PID_Status();
R_TRIG_0(CLK := PID.MODE.eMode=ePID_Modes.Auto); // R_trig
IF R_TRIG_0.Q THEN _w1 := PID.HMI_Target; END_IF
PID.PLC_Target := _w1;
_w2 := SEL(PID.MODE.eMode=ePID_Modes.Auto, PId.HMI_Target, PID.PLC_Target);
PID.Live_Target := _w2;
_w3 := _w2 * PID.FF;
PID.CV_FF := _w3;
_w4 := SEL(Reverse, _w2 - PID.Actual, PID.Actual - _w2);
PID.Err := _w4;
_w5 := SEL(PID.MODE.eMode=ePID_Modes.Auto, PID.MODE.eMode=ePID_Modes.FORCED_ON, PID.PLC_Enable AND (Not(PID.Inhibit))) AND True AND CV_OK AND PV_OK;
Loop_Enable := _w5;
FT_PIDW_0(
    IN := _w4,
    KP := PID.KP,
    TN := PID.TN,
    TV := PID.TV,
    LIM_L := PID.CV_Min-PID.CV_FF,
    LIM_H := PID.CV_Max-PID.CV_FF,
    RST := R_Trig_1.Q OR NOT _w5); // BURKERT_OSCAT_BASIC.FT_PIDW
_w6 := SEL(Loop_Enable, PID.CV_Min, _w3 + FT_PIDW_0.Y);
CV := _w6;
PID.CV := _w6;
PID.CV_P := PID.Err * PID.KP;
PID.CV_I := FT_PIDW_0.YI;
PID.CV_D := FT_PIDW_0.diff.out;
PID.Ready := (PID.MODE.eMode=ePID_Modes.Auto) AND CV_OK AND PV_OK;
R_TRIG_1(CLK := (PID.CV_P>0) AND (PID.CV_I<0) AND (FT_PIDW_0.Y<0.5) AND _w5); // R_Trig
IF NOT (PID.MODE.eMode=ePID_Modes.FORCED_ON) THEN _w7 := PID.PLC_Target; END_IF
PID.HMI_Target := _w7;

END_FUNCTION_BLOCK

// 20 Program Organization Units/Level_2_Controls/Quick_Mix_UDFB
FUNCTION_BLOCK Quick_Mix_UDFB
VAR_INPUT
	Destination_OK:BOOL;
END_VAR
VAR_OUTPUT
	//Active:BOOL;
	OK:BOOL;
END_VAR
VAR
	Current_Mode:eQuick_Mix_modes;
	Current_Status:eQuick_Mix_Status;
	SFCReset:BOOL;
	SFCInit:BOOL;
	PLC_Active:BOOL;
	Temp_PID:BURKERT_OSCAT_BASIC.FT_PIDW;
	Flow_PID:BURKERT_OSCAT_BASIC.FT_PIDW;
	Ramp:Burkert_OSCAT_BASIC.SRAMP;
	tRamp:Burkert_OSCAT_BASIC.SRAMP;
	Ramp_Time:TIME;
	Pause_Active:BOOL;
	Pause_Ton:Ton;
	//Temp_Control:Burkert_OSCAT_BASIC.SCALE_R;
	//Flow_Control:Burkert_OSCAT_BASIC.SCALE_R;
	tHW:REAL;
END_VAR
VAR_IN_OUT
	HW:cACV;
	CW:cACV;
	FIT:cFIT;
	TT:cAIT;
	Loop:Quick_Mix_Dut;
END_VAR

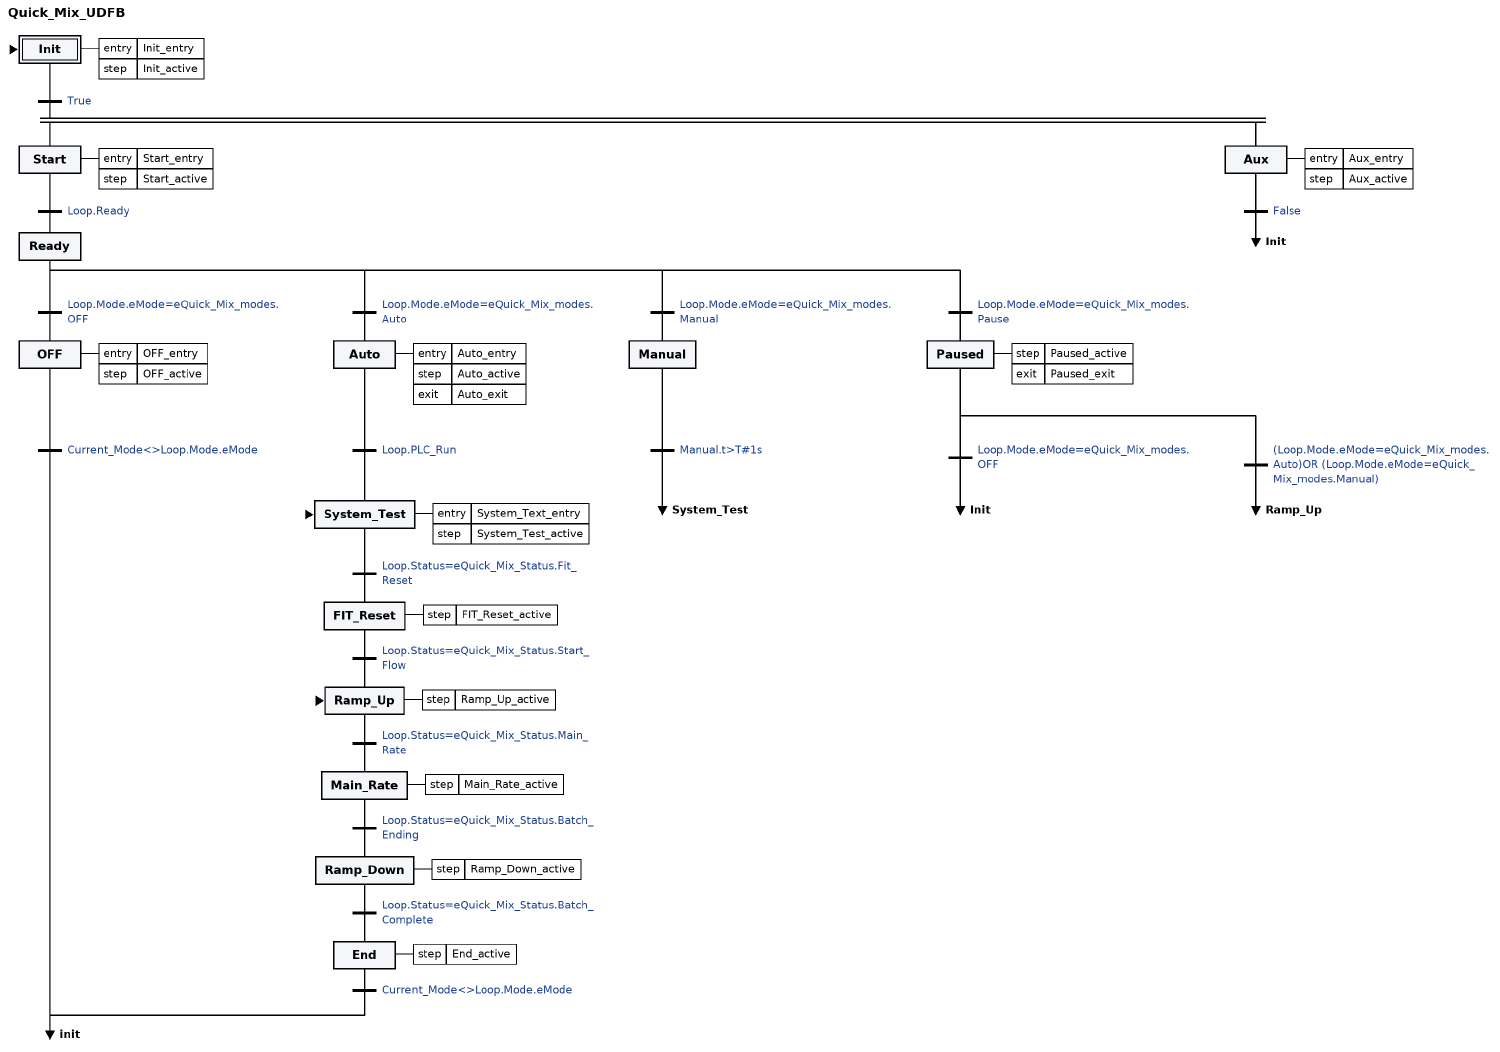
INITIAL_STEP Init:
    Init_entry(P1);  // entry action
    Init_active(N);  // step action
END_STEP
TRANSITION FROM Init TO (Start, Aux)
    := True;
END_TRANSITION
STEP Start:
    Start_entry(P1);  // entry action
    Start_active(N);  // step action
END_STEP
TRANSITION FROM Start TO Ready
    := Loop.Ready;
END_TRANSITION
STEP Ready:
END_STEP
STEP Aux:
    Aux_entry(P1);  // entry action
    Aux_active(N);  // step action
END_STEP
TRANSITION FROM Aux TO Init
    := False;
END_TRANSITION
TRANSITION FROM Ready TO OFF
    := Loop.Mode.eMode=eQuick_Mix_modes.OFF;
END_TRANSITION
STEP OFF:
    OFF_entry(P1);  // entry action
    OFF_active(N);  // step action
END_STEP
TRANSITION FROM OFF TO init
    := Current_Mode<>Loop.Mode.eMode;
END_TRANSITION
TRANSITION FROM Ready TO Auto
    := Loop.Mode.eMode=eQuick_Mix_modes.Auto;
END_TRANSITION
STEP Auto:
    Auto_entry(P1);  // entry action
    Auto_active(N);  // step action
    Auto_exit(P0);  // exit action
END_STEP
TRANSITION FROM Auto TO System_Test
    := Loop.PLC_Run;
END_TRANSITION
STEP System_Test:
    System_Text_entry(P1);  // entry action
    System_Test_active(N);  // step action
END_STEP
TRANSITION FROM System_Test TO FIT_Reset
    := Loop.Status=eQuick_Mix_Status.Fit_Reset;
END_TRANSITION
STEP FIT_Reset:
    FIT_Reset_active(N);  // step action
END_STEP
TRANSITION FROM FIT_Reset TO Ramp_Up
    := Loop.Status=eQuick_Mix_Status.Start_Flow;
END_TRANSITION
STEP Ramp_Up:
    Ramp_Up_active(N);  // step action
END_STEP
TRANSITION FROM Ramp_Up TO Main_Rate
    := Loop.Status=eQuick_Mix_Status.Main_Rate;
END_TRANSITION
STEP Main_Rate:
    Main_Rate_active(N);  // step action
END_STEP
TRANSITION FROM Main_Rate TO Ramp_Down
    := Loop.Status=eQuick_Mix_Status.Batch_Ending;
END_TRANSITION
STEP Ramp_Down:
    Ramp_Down_active(N);  // step action
END_STEP
TRANSITION FROM Ramp_Down TO End
    := Loop.Status=eQuick_Mix_Status.Batch_Complete;
END_TRANSITION
STEP End:
    End_active(N);  // step action
END_STEP
TRANSITION FROM End TO init
    := Current_Mode<>Loop.Mode.eMode;
END_TRANSITION
TRANSITION FROM Ready TO Manual
    := Loop.Mode.eMode=eQuick_Mix_modes.Manual;
END_TRANSITION
STEP Manual:
END_STEP
TRANSITION FROM Manual TO System_Test
    := Manual.t>T#1s;
END_TRANSITION
TRANSITION FROM Ready TO Paused
    := Loop.Mode.eMode=eQuick_Mix_modes.Pause;
END_TRANSITION
STEP Paused:
    Paused_active(N);  // step action
    Paused_exit(P0);  // exit action
END_STEP
TRANSITION FROM Paused TO Init
    := Loop.Mode.eMode=eQuick_Mix_modes.OFF;
END_TRANSITION
TRANSITION FROM Paused TO Ramp_Up
    := (Loop.Mode.eMode=eQuick_Mix_modes.Auto)OR (Loop.Mode.eMode=eQuick_Mix_modes.Manual);
END_TRANSITION

END_FUNCTION_BLOCK

// 20 Program Organization Units/Level_2_Controls/Rate_Batch
FUNCTION_BLOCK Rate_Batch
VAR_INPUT
	Config: REFERENCE TO cBatch;
	Rate_PID:	REFERENCE TO PID_Control;
	Volume_PID:	REFERENCE TO PID_Control;
	FIT:	REFERENCE TO cFIT;
	
	CV_OK:BOOL;
END_VAR
VAR_OUTPUT
	CV:REAL;
END_VAR
VAR
	Local_Mode:eHOA_Modes;
	Local_Task:eBatch_Task;
	Local_Status:eBatch_Status;
	
	Start_Rate:REAL;
	Main_Rate:REAL;
	End_Rate:REAL;
	
	
	Batch_Duration_S:UINT;
	clk_250:Burkert_OSCAT_BASIC.CLK_PRG;
	Batch_Clock_S:REAL;
	
END_VAR

CASE Config.Mode.eMode OF
	eHOA_Modes.Off:		Mode_OFF();
	eHOA_Modes.Manual:	Mode_Manual();
	eHOA_Modes.Auto:	Mode_Auto();	
END_CASE


CASE Config.Task OF
	eBatch_task.OFF	: 	Task_OFf();
	eBatch_task.Pause :	Task_Pause();
	eBatch_Task.Resume: Task_Resume();
	eBatch_task.Run:	Task_Run();
END_CASE

END_FUNCTION_BLOCK

// 20 Program Organization Units/Level_2_Controls/SSR_Heater
FUNCTION_BLOCK SSR_Heater
VAR_INPUT
	Heater: REFERENCE TO cSSR_heater;
	CV:REAL;
END_VAR
VAR_OUTPUT
	
END_VAR
VAR
	//Output_CV:UINT;
	CV_Error:REAL;
	//Output_Base:UINT;
	//Output_Map:WORD;
	
	SRR_1_U_CTRL:OSCAT_BUILDING.ACTUATOR_PUMP;
	SRR_1_V_CTRL:OSCAT_BUILDING.ACTUATOR_PUMP;
	SRR_1_W_CTRL:OSCAT_BUILDING.ACTUATOR_PUMP;
	
	SRR_2_U_CTRL:OSCAT_BUILDING.ACTUATOR_PUMP;
	SRR_2_V_CTRL:OSCAT_BUILDING.ACTUATOR_PUMP;
	SRR_2_W_CTRL:OSCAT_BUILDING.ACTUATOR_PUMP;
	
	SRR_3_U_CTRL:OSCAT_BUILDING.ACTUATOR_PUMP;
	SRR_3_V_CTRL:OSCAT_BUILDING.ACTUATOR_PUMP;
	SRR_3_W_CTRL:OSCAT_BUILDING.ACTUATOR_PUMP;
	
	Main_Contactor: RS;
	Force_Group_Sort:Bool;
	Group_Sorted:BOOL;
	Group_Sort_Array:ARRAY[0..2] OF REAL;
	Group_Sort_Index:ARRAY[0..2] OF INT;
	

	Pulse_30Min:Burkert_OSCAT_BASIC.CLK_PRG;
	CV_Index:INT:=0;
	Ramp:util.RAMP_REAL;
END_VAR

(*

0%			ALL OFF
11%			Single Pair
22%			2 Single Pair 
33%			Double Pair Full SSR
44%			Double Pair plus Single
55%			Double Pair Plus 2 Single Pairs
66%			2 Double Pair Full SSR
77%			Double Pair Full SSR + Single Pair
88%			
99%			All SSR's
*)



Select_CV();
Pulse_30Min(PT:=T#30M);
IF Pulse_30Min.Q OR Force_Group_Sort THEN
	Sort_Groups();
END_IF;

Set_Ouputs();

//Outputs();

SSR_Control();

RAMP( 
	ASCEND:= 10, 
	DESCEND:= 10, 
	TIMEBASE:= T#10S, 
	RESET:= , 
	OUT=>Heater.Effective_Output );

END_FUNCTION_BLOCK

// 20 Program Organization Units/Level_2_Controls/Stack_Lights_4Way
FUNCTION_BLOCK Stack_Lights_4Way
VAR_INPUT
END_VAR
VAR_OUTPUT
	Red:BOOL;
	Yellow:BOOL;
	Green:BOOL;
	Horn:BOOL;
	
END_VAR
VAR
	
	GEN_PULSE_RED: Burkert_OSCAT_BASIC.GEN_PULSE;
	GEN_PULSE_Yellow: Burkert_OSCAT_BASIC.GEN_PULSE;
	GEN_PULSE_Green: Burkert_OSCAT_BASIC.GEN_PULSE;
	GEN_PULSE_Horn: Burkert_OSCAT_BASIC.GEN_PULSE;
END_VAR

VAR_IN_out
	Device:c4Way_Stack_Light;
END_VAR
VAR // added by the converter: edge detectors and wires of the graphical bodies
    _w1, _w2, _w3, _w4 : ANY;
END_VAR

GEN_PULSE_Yellow(
    ENQ := Device.Yellow.Flash_Rate_ms>500 AND Device.Yellow.ON,
    PTH := To_Time(Device.Yellow.Flash_Rate_ms),
    PTL := To_Time(Device.Yellow.Flash_Rate_ms)); // Burkert_OSCAT_BASIC.GEN_PULSE
GEN_PULSE_Green(
    ENQ := Device.Green.Flash_Rate_ms>500 AND Device.Green.ON,
    PTH := To_Time(Device.Green .Flash_Rate_ms),
    PTL := To_Time(Device.Green .Flash_Rate_ms)); // Burkert_OSCAT_BASIC.GEN_PULSE
GEN_PULSE_Horn(
    ENQ := Device.Horn.Flash_Rate_ms>500 AND Device.Horn.ON,
    PTH := To_Time(Device.Horn .Flash_Rate_ms),
    PTL := To_Time(Device.Horn .Flash_Rate_ms)); // Burkert_OSCAT_BASIC.GEN_PULSE
_w1 := Device.Horn.ON AND NOT GEN_PULSE_Horn.Q;
Horn := _w1;
_w2 := Device.Yellow.ON AND NOT GEN_PULSE_Yellow.Q;
Device.Yellow.Q := _w2;
Yellow := _w2;
_w3 := Device.Green.ON AND NOT GEN_PULSE_Green.Q;
Device.Green.Q := _w3;
Green := _w3;
GEN_PULSE_RED(
    ENQ := Device.RED.Flash_Rate_ms>500 AND Device.RED.ON,
    PTH := To_Time(Device.RED.Flash_Rate_ms),
    PTL := To_Time(Device.RED.Flash_Rate_ms)); // Burkert_OSCAT_BASIC.GEN_PULSE
_w4 := Device.RED.ON AND NOT GEN_PULSE_RED.Q;
Device.RED.Q := _w4;
Red := _w4;
Device.Horn.Q := _w1;

END_FUNCTION_BLOCK

// 20 Program Organization Units/Level_2_Controls/SW_CTRL
FUNCTION_BLOCK SW_CTRL 
VAR_INPUT
	SW: REFERENCE TO cBatch_Transfer;
	FIT:REFERENCE TO cFIT;
	BCV:REFERENCE TO cBCV;
	Pump_Ready:BOOL;
	Interlock:BOOL;
END_VAR
VAR
	PID: BURKERT_OSCAT_BASIC.FT_PIDW;
END_VAR

IF (
		((SW.Auto_Batch = FALSE AND SW.Mode.eMode=eBatch_Transfer_Mode.Auto) OR
		(SW.Mode.eMode=eBatch_Transfer_Mode.Disabled)) AND SW.Status<> Transfer_Status.IDLE
	) THEN
	SW.Status:=Transfer_Status.IDLE;
END_IF;

IF (FIT.Rate.EU>1 AND NOT(BCV.Status.eStatus=eBCV_Status.A_Open) AND NOT(Interlock)) THEN
	SW.Status:=Transfer_Status.Flow_Meter_Active;
	SW.Ready:=FALSE;
	SW.Active:=FALSE;
END_IF;

IF NOT(Pump_Ready) THEN
	SW.Status:=Transfer_Status.Pump_Not_Ready;
	SW.Ready:=FALSE;
	SW.Active:=FALSE;
END_IF


IF NOT(BCV.Ready) THEN
	SW.Status:=Transfer_Status.BCV_Not_Ready;
	SW.Ready:=FALSE;
	SW.Active:=FALSE;
END_IF;

IF (BCV.Status.eStatus=eBCV_Status.Interlocked OR BCV.Status.eStatus=eBCV_Status.LOCKED_OUT ) THEN
	SW.Status:=Transfer_Status.LOCKED_OUT;
	SW.Ready:=FALSE;
	SW.Active:=FALSE;
END_IF;


IF Sw.Status=Transfer_Status.IDLE AND Interlock THEN
	SW.Status:=Transfer_Status.LOCKED_OUT;
END_IF

CASE SW.Status OF
	
	Transfer_Status.IDLE:
		SW.Ready:=TRUE;
		SW.BCV:=FALSE;
		
		SW.Remaining_Time_S:=0;
		SW.Current_Rate:=0;
		SW.Current_Volume:=0;
		SW.Remaining_Volume:=0;
		SW.Active:=FALSE;
		
		IF (
			(SW.Auto_Batch AND SW.Mode.eMode=eBatch_Transfer_Mode.Auto) OR
			( SW.Mode.eMode=eBatch_Transfer_Mode.Batch)
			)THEN
			SW.Status:=Transfer_Status.FIT_Reset;
		END_IF;
		
		
	Transfer_Status.FIT_Reset:
		SW.Active:=TRUE;
		SW.BCV:=FALSE;
		SW.Remaining_Time_S:=0;
		FIT.PLC_Reset:=(FIT.Total>1);
		IF FIT.Total<1 THEN
			SW.Status:=Transfer_Status.Open_Valve;
		END_IF;
		
	Transfer_Status.Open_Valve:
	SW.BCV:=TRUE;
	IF SW.BCV AND BCV.Status.eStatus=eBCV_Status.A_Open THEN
			SW.Status:=Transfer_Status.Flow_Active;	
		END_IF;
		
	
		
	Transfer_Status.Flow_Active:
		SW.BCV:=TRUE;
		SW.Remaining_Time_S:=TO_UDINT(SW.Remaining_Volume/(FIT.Rate.EU/60));
		SW.Current_Rate:=FIT.Rate.EU;
		SW.Current_Volume:=FIT.Total;
		SW.Remaining_Volume:=(SW.Volume-FIT.Total);
		
		
		IF (
			(FIT.Rate.EU > (SW.Rate*0.25)) OR
			(FIT.Total> (SW.Volume*0.80))
		) THEN
			SW.Status:=Transfer_Status.Running;
		END_IF;
	Transfer_Status.Running:	
			SW.BCV:=TRUE;
			SW.Remaining_Time_S:=TO_UDINT(SW.Remaining_Volume/(FIT.Rate.EU/60));
			SW.Current_Rate:=FIT.Rate.EU;
			SW.Current_Volume:=FIT.Total;	
			SW.Remaining_Volume:=(SW.Volume-FIT.Total);
			IF (FIT.Total> SW.Volume)
			THEN
				SW.Status:=Transfer_Status.Complete;
			END_IF;
	Transfer_Status.Complete:
		SW.BCV:=FALSE;
		SW.Remaining_Time_S:=0;
		SW.Current_Rate:=0;
		SW.Current_Volume:=0;
		SW.Remaining_Volume:=0;
		SW.Active:=FALSE;
		
	Transfer_Status.LOCKED_OUT:
		SW.Ready:=FALSE;
		SW.Active:=FALSE;
		SW.Remaining_Time_S:=0;
		SW.Current_Rate:=0;
		SW.Current_Volume:=0;
		SW.Remaining_Volume:=0;
		
		
	Transfer_Status.Destination_Not_Ready:
		SW.Active:=FALSE;
		IF SW.BCV AND BCV.Status.eStatus=eBCV_Status.A_Open THEN
			SW.Status:=Transfer_Status.Flow_Active;		
		END_IF;
		IF 	(
				NOT(SW.Mode.eMode=eBatch_Transfer_mode.Auto AND SW.Auto_Batch = TRUE) AND
				NOT(SW.Mode.eMode=eBatch_Transfer_mode.Batch) AND
				SW.BCV=TRUE
			)THEN
			SW.BCV:=FALSE;
		END_IF;
	Transfer_Status.Flow_Meter_Active:
		IF FIT.Rate.EU<0.5 THEN
			SW.Status:=Transfer_Status.IDLE;
		END_IF;
END_CASE;



PID(
	IN:= (SW.Rate-FIT.Rate.EU), 
	KP:= SW.Config.KP, 
	TN:= SW.Config.TN, 
	TV:= SW.Config.TV, 
	LIM_L:= 0, 
	LIM_H:= 100-(SW.Config.FF*SW.Rate), 
	RST:= NOT(SW.Active) OR NOT(BCV.Status.eStatus=eBCV_Status.A_Open) , 
	Y=> , 
	LIM=> );
	
IF NOT(SW.Active) THEN
	SW.ACV:=0;
	SW.BCV:=FALSE;
ELSE
	SW.ACV:=PID.Y+(SW.Config.FF*SW.Rate);

END_IF;

END_FUNCTION_BLOCK

// 20 Program Organization Units/Level_2_Controls/Tempered_Line_4_Valve
FUNCTION_BLOCK Tempered_Line_4_Valve
VAR_INPUT
	Config_DATA:REFERENCE TO cTempered_Line_Data;
	
	HW_Supply_TT:REFERENCE TO cSensor;
	CW_Supply_TT:REFERENCE TO cSensor;
	
	CW_Inlet_PT:REFERENCE TO cSensor;
	CW_Outlet_PT:REFERENCE TO cSensor;
	HW_Inlet_PT:REFERENCE TO cSensor;
	HW_Outlet_PT:REFERENCE TO cSensor;
	Combined_Temp:REFERENCE TO cSensor;
	
	HW_FIT:REFERENCE TO cFIT;
	CW_FIT:REFERENCE TO cFIT;

	HW_PID		:REFERENCE TO PID_DUT;
	CW_PID		:REFERENCE TO PID_DUT;
	Temperature_PID		:REFERENCE TO PID_DUT;
	
	CW1_ACV		:REFERENCE TO cACV;
	CW2_ACV		:REFERENCE TO cACV;
	HW1_ACV		:REFERENCE TO cACV;
	HW2_ACV		:REFERENCE TO cACV;
	
	KV_Curve	:REFERENCE TO ARRAY[0..100] OF REAL;
	CV_2_KV		:REFERENCE TO ARRAY[0..100] OF REAL;
	
	Temp_Flow_CV	:REFERENCE TO cTempered_C;
	
	Flow_Units:eUnits;
	Temperature_Units:eUnits;
	Run_mode:BYTE;
	
	
	HW_CV_Mode_3:INT;
	CW_CV_Mode_3:INT;
	
END_VAR
VAR_OUTPUT
END_VAR
VAR
	Local_Mode:eTempered_modes;
	Local_Task:eTempered_Task;
	Local_Status:eTempered_Status;
	On_Target:BOOL;
	Task_Ton:Ton;
	Prepare_TON:TON;
	
	
	Temp_Index:INT;
	Flow_Index:INT;
	
	CW_KV_Index:INT;
	HW_KV_Index:INT;
	
	CW_Target_KV_Index:INT;
	HW_Target_KV_Index:INT;
	
	Calibration_Temp:cAlarm_Window;
	
	
	KV_Index_Scalar:INT:=20;
	
	HW_CV_Ramp:RAMP_REAL;
	CW_CV_Ramp:RAMP_REAL;
	
	TOF_0: TOF;
END_VAR

AUX();
Alarms();
Math();
PID_CTRL();
ACV_CTRL();

Task_Ton();

END_FUNCTION_BLOCK

// 20 Program Organization Units/Level_2_Controls/Tempered_Mix_UDFB
FUNCTION_BLOCK Tempered_Mix_UDFB
VAR_INPUT
	//Loop_ID:INT;
END_VAR
VAR_IN_OUT
	HW_ACV:cACV;
	CW_ACV:cACV;
	Temperature:cAIT;
	FIT:cFIT;
	Control:Mix_DUT;
END_VAR
VAR_OUTPUT
END_VAR
VAR
	R_TRIG_0: R_Trig;
	RATE_PID: BURKERT_OSCAT_BASIC.CTRL_PID;
	
	Temp_PID: BURKERT_OSCAT_BASIC.CTRL_PID;
	TON_0: TON;
	Stage_Delay: TIME := T#2s;
	TON_1: TON;
	TON_2: TON;
	SRAMP_0: BURKERT_OSCAT_BASIC.SRAMP;
	TON_3: TON;
	TON_4: TON;
	Ramp_Active: BOOL;
	Ramp_Target: REAL;
	TON_5: TON;
	TON_6: TON;
	R_TRIG_1: R_trig;
	Ramp_Start_Volume: REAL;
	Ramp_Volume: REAL;
	R_TRIG_2: R_Trig;
	R_TRIG_3: R_Trig;
	PID_0: Util.PID;
	R_TRIG_4: R_Trig;
	R_TRIG_5:R_trig;
	
	Live_Rate: REAL;
END_VAR
VAR // added by the converter: edge detectors and wires of the graphical bodies
    _w1, _w2, _w3, _w4, _w5, _w6, _w10, _w12, _w13, _w14, _w15, _w16, _w18, _w19, _w21, _w23, _w25, _w30, _w32 : ANY;
    _w7, _w8, _w9, _w11, _w17, _w20, _w22, _w24, _w26, _w28, _w29, _w31, _w33 : BOOL;
    _w27 : REAL;
END_VAR

// note: 18 stored wires end on pins the file does not list and are not shown
IF NOT (HW_ACV.Mode.eMode=eACV_Modes.Auto) THEN _w1 := Mix_Status.HW_Valve_Not_Ready; END_IF
Control.Status := _w1;
IF NOT (CW_ACV.Mode.eMode=eACV_Modes.Auto) THEN _w2 := Mix_Status.CW_Valve_Not_Ready; END_IF
Control.Status := _w2;
Control.Actual_Rate_EU := FIT.Rate.EU;
_w3 := (Control.Mode=Mix_Modes.IDlE) OR (Control.STATUS>Mix_Status.Batch_Ending) OR (Control.Mode=Mix_Modes.Pause);
RATE_PID(
    ACT := FIT.Rate.EU,
    SET := Live_Rate,
    SUP := 0.1,
    OFS := 0.0,
    M_I := 0.0,
    MAN := _w3,
    RST := _w3,
    KP := Control.Config.Flow_KP,
    TN := Control.Config.Flow_TN,
    TV := Control.Config.Flow_TV,
    LL := 0,
    LH := 100.0); // BURKERT_OSCAT_BASIC.CTRL_PID
Control.Flow_CV := RATE_PID.Y;
R_TRIG_2(CLK := _w3 AND (Temperature.Mode.eMode<>AIT_Modes.Forced)); // R_Trig
IF R_TRIG_2.Q THEN _w4 := AIT_Modes.Alarms_Disabled; END_IF
Temperature.Mode.eMode := _w4;
Control.Actual_Temp_EU := Temperature.EU;
_w5 := (Control.Mode=Mix_Modes.IDlE) OR (Control.Mode=Mix_Modes.Rate_Only) OR (Control.STATUS>Mix_Status.Batch_Ending) OR (Control.STATUS=Mix_Status.Start_Flow) OR (Control.STATUS=Mix_Status.Fit_Reset) OR (Control.Mode=Mix_Modes.Pause);
PID_0(
    ACTUAL := Temperature.EU,
    SET_POINT := Control.Config.TARGET_C,
    KP := Control.Config.Temp_KP,
    TN := Control.Config.Temp_TN,
    TV := Control.Config.Temp_TV,
    Y_MANUAL := 0,
    Y_OFFSET := 0,
    Y_MIN := -100,
    Y_MAX := 100,
    MANUAL := _w5,
    RESET := _w5); // Util.PID
Control.Temp_CV := SEl(Control.Mode=Mix_Modes.Cold_Only, SEl(Control.Mode=Mix_Modes.Hot_Only, PID_0.Y, 100), -100);
SRAMP_0(
    X := Ramp_Target,
    A_UP := Control.Config.Ramp_Rate,
    A_DN := 0-Control.config.Ramp_Rate,
    VU_MAX := Control.config.Max_Flow,
    VD_MAX := 0-Control.config.Max_Flow,
    LIMIT_HIGH := Control.config.Max_Flow,
    LIMIT_LOW := Control.Config.Min_Flow,
    RST := Control.Mode=Mix_Modes.IDlE); // BURKERT_OSCAT_BASIC.SRAMP
Live_Rate := SRAMP_0.Y;
IF Control.Mode=Mix_Modes.IDlE THEN _w6 := Mix_Status.IDle; END_IF
Control.STATUS := _w6;
R_TRIG_0(CLK := (Control.Mode=Mix_Modes.Auto) OR (Control.Mode=Mix_Modes.Hot_Only) OR (Control.Mode=Mix_Modes.Cold_Only) OR (Control.Mode=Mix_Modes.Quick_Start)); // R_Trig
Control.STATUS := SEL(R_TRIG_0.Q, Control.STATUS, Mix_Status.Fit_Reset);
Control.Actual_Volume_EU := FIT.Total;
_w7 := Control.STATUS = Mix_Status.Fit_Reset;
_w8 := NOT (FIT.Total>0.1) AND _w7;
FIT.PLC_Reset := SEL(_w7 AND (FIT.Total>0.1), SEL(_w8, FIT.PLC_Reset, False), True);
_w9 := _w8;
IF _w9 THEN _w10 := Mix_Status.Start_Flow; END_IF
_w11 := _w9;
IF _w11 THEN _w12 := SEL(Control.Mode=Mix_Modes.Hot_Only, _w10, Mix_Status.Temperature_OK); END_IF
IF _w11 THEN _w13 := SEL(Control.Mode=Mix_Modes.Hot_Only, _w12, Mix_Status.Temperature_OK); END_IF
Control.STATUS := _w13;
_w14 := Control.Temp_CV / 100.0;
_w15 := LIMIT(0, Control.Flow_CV * (1.0 + _w14), 100);
Control.HW_CMD := _w15;
HW_ACV.PLC_CMD := _w15;
_w16 := LIMIT(0, Control.Flow_CV * (1.0 - _w14), 100);
Control.CW_CMD := _w16;
CW_ACV.PLC_CMD := _w16;
_w17 := Control.STATUS = Mix_Status.Start_Flow;
IF _w17 THEN _w18 := Control.Config.Min_Flow; END_IF
Ramp_Target := _w18;
TON_0(IN := _w17 AND (Control.Actual_Rate_EU > (Control.Config.Min_Flow*0.8) OR (Control.Mode=Mix_Modes.Quick_Start)), PT := Stage_Delay); // TON
Control.STATUS := SEL(TON_0.Q, Control.STATUS, Mix_Status.Flow_Detected);
TON_1(IN := Control.STATUS = Mix_Status.Flow_Detected, PT := Stage_Delay); // TON
R_TRIG_3(CLK := (Temperature.Mode.eMode<>AIT_Modes.Forced) AND TON_1.Q); // R_Trig
IF R_TRIG_3.Q THEN _w19 := TT_Modes.Active; END_IF
Temperature.Mode.iMode := _w19;
Control.STATUS := SEL(TON_1.Q, Control.STATUS, Mix_Status.Start_temperature);
Temperature.Alarm_Config.Setpoints.Hi_Hi_Alarm := Control.Config.TARGET_C+(Control.Config.TEMP_WINDOW*4);
Temperature.Alarm_Config.Setpoints.Hi_Warn := Control.Config.TARGET_C+(Control.Config.TEMP_WINDOW*2);
Temperature.Alarm_Config.Setpoints.Low_warn := Control.Config.TARGET_C-(Control.Config.TEMP_WINDOW*2);
Temperature.Alarm_Config.Setpoints.Low_Low_Alarm := Control.Config.TARGET_C-(Control.Config.TEMP_WINDOW*4);
TON_2(IN := Control.STATUS = Mix_Status.Start_temperature AND (Control.Actual_Temp_EU > (Control.Config.TARGET_C-Control.Config.TEMP_WINDOW) OR (Control.Mode=Mix_Modes.Quick_Start)), PT := Stage_Delay); // TON
Control.STATUS := SEL(TON_2.Q, Control.STATUS, Mix_Status.Temperature_OK);
TON_3(IN := Control.STATUS = Mix_Status.Temperature_OK, PT := Stage_Delay); // TON
Control.STATUS := SEL(TON_3.Q, Control.STATUS, Mix_Status.Foundation_Rate);
_w20 := Control.STATUS = Mix_Status.Foundation_Rate;
IF _w20 THEN _w21 := Control.Config.Foundation_Rate; END_IF
Ramp_Target := _w21;
Control.STATUS := SEL(_w20 AND (Control.Actual_Rate_EU >= (Control.Config.Foundation_Rate*0.9) OR (Control.Mode=Mix_Modes.Quick_Start)), Control.STATUS, Mix_Status.Foundation_Rate_OK);
TON_4(IN := Control.STATUS = Mix_Status.Foundation_Rate_OK AND (FIT.Total >= Control.Config.Foundation_Volume OR (Control.Mode=Mix_Modes.Quick_Start)), PT := Stage_Delay); // TON
Control.STATUS := SEL(TON_4.Q, Control.STATUS, Mix_Status.Foundation_Amount_Complete);
R_TRIG_5(CLK := Control.Mode=Mix_Modes.Resume); // R_trig
TON_5(IN := Control.STATUS = Mix_Status.Foundation_Amount_Complete, PT := Stage_Delay); // TON
Control.STATUS := SEL(R_TRIG_5.Q OR TON_5.Q, Control.STATUS, Mix_Status.Main_Rate);
_w22 := Control.STATUS = Mix_Status.Main_Rate;
R_TRIG_1(CLK := _w22); // R_trig
IF R_TRIG_1.Q THEN _w23 := Control.Actual_Volume_EU; END_IF
Ramp_Start_Volume := _w23;
_w24 := _w22;
IF _w24 THEN _w25 := Control.Config.TARGET_lpm; END_IF
Ramp_Target := _w25;
_w26 := _w24 AND Control.Actual_Rate_EU >= (Control.Config.TARGET_lpm*0.9);
Control.STATUS := SEL(_w26, Control.STATUS, Mix_Status.Main_Rate_OK);
IF _w26 THEN _w27 := Control.Actual_Volume_EU - Ramp_Start_Volume; END_IF
Ramp_Volume := _w27;
_w28 := Control.STATUS = Mix_Status.Main_Rate_OK;
TON_6(IN := _w28, PT := Stage_Delay); // TON
Control.STATUS := SEL(TON_6.Q, Control.STATUS, Mix_Status.Grain_Dispense);
_w29 := Control.STATUS = Mix_Status.Grain_Dispense;
IF _w29 THEN _w30 := Control.Config.TARGET_lpm; END_IF
Ramp_Target := _w30;
Control.STATUS := SEL(_w29 AND Control.Actual_Volume_EU >= (Control.Config.TARGET_L-Control.Config.Foundation_Volume), Control.STATUS, Mix_Status.Batch_Ending);
Control.Grain_ETA_S := REAL_TO_INT(((Control.Config.TARGET_L-Control.Config.Foundation_Volume) - Control.Actual_Volume_EU) / (Control.Actual_Rate_EU/60));
_w31 := Control.STATUS = Mix_Status.Batch_Ending;
IF _w31 THEN _w32 := Control.Config.Foundation_Rate; END_IF
Ramp_Target := _w32;
_w33 := (_w22 OR _w28 OR _w29 OR _w31) AND Control.Actual_Volume_EU >= Control.Config.TARGET_L;
Ramp_Active := SEl(_w33, Ramp_Active, FALSE);
Control.STATUS := SEL(_w33, Control.STATUS, Mix_Status.Batch_Complete);
// 0.1: input not connected

END_FUNCTION_BLOCK

// 20 Program Organization Units/Simulators/c8691_CanOpen_Sim
FUNCTION_BLOCK cDigital_BCV_CanOpen_Sim
VAR_INPUT
	BCV: REFERENCE TO cDigital_BCV;
END_VAR
VAR_OUTPUT
END_VAR
VAR
END_VAR

BCV.PDO.EndPositions.1:=BCV.PDO.Setpoint.0;
BCV.PDO.EndPositions.0:=NOT(BCV.PDO.Setpoint.0);
BCV.PDO.NamurStatus:=1;

END_FUNCTION_BLOCK

// 20 Program Organization Units/Simulators/c8694_CanOpen_Sim
FUNCTION cDigital_ACV_CanOpen_Sim
VAR_INPUT
END_VAR
VAR_OUTPUT
	//CanState:_3SCOS.DED.DEVICE_STATE;
END_VAR
VAR
	//Data:Bytes_Dword;
END_VAR
VAR_IN_OUT
	Device:cCanOpen_8694;
END_VAR


Device.PDO.NamurStatus:=1;

Device.PDO.CMD:=Device.PDO.CMDdigital;
Device.PDO.Pos:=Device.PDO.CMDdigital;

//CanState:=_3SCOS.DED.DEVICE_STATE.RUNNING;


Device.CanOpen.Device_State:=_3SCOS.DED.DEVICE_STATE.RUNNING;

END_FUNCTION

// 20 Program Organization Units/Simulators/CalculateMixedConductivity
FUNCTION CalculateMixedConductivity : Real
VAR_INPUT
    Stream_A_Rate        : REAL;  (* Flow rate of Stream A in liters per minute *)
    Stream_A_Conductivity: REAL;  (* Conductivity of Stream A in µS/cm *)
    Stream_B_Rate        : REAL;  (* Flow rate of Stream B in liters per minute *)
    Stream_B_Conductivity: REAL;  (* Conductivity of Stream B in µS/cm *)
END_VAR
VAR
    TotalFlowRate       : REAL;
    WeightedConductivity: REAL;
END_VAR

IF Stream_A_Rate>0.05 AND Stream_B_Rate>0.05 THEN
    TotalFlowRate := Stream_A_Rate + Stream_B_Rate;
    WeightedConductivity := ((Stream_A_Conductivity * Stream_A_Rate) + (Stream_B_Conductivity * Stream_B_Rate)) / TotalFlowRate;
    CalculateMixedConductivity := WeightedConductivity;
ELSE
	CalculateMixedConductivity :=MIN(Stream_A_Conductivity,Stream_B_Conductivity);
END_IF;

END_FUNCTION

// 20 Program Organization Units/Simulators/CanOpen_8694_Data_Sim
FUNCTION CanOpen_8694_Data_Sim
VAR_INPUT
END_VAR
VAR_OUTPUT
END_VAR
VAR
	//Data:Bytes_Dword;
END_VAR
VAR_IN_OUT
	Device:cCanOpen_8694;
END_VAR



Device.PDO.NamurStatus:=1;
Device.PDO.Pos:=Device.PDO.CMDdigital;
Device.CanOpen.Device_State:=_3SCOS.DED.DEVICE_STATE.DISABLED;

END_FUNCTION

// 20 Program Organization Units/Simulators/Contactor_Sim
FUNCTION_BLOCK Contactor_Sim
VAR_INPUT
	Device:Contactor_DUT;
END_VAR
VAR_OUTPUT
	FWD_Limit:BOOL;
	Rev_Limit:BOOL;
END_VAR
VAR
	tPos:INT;
	pulse: Burkert_OSCAT_BASIC.CLK_PRG;
END_VAR

Pulse(PT:=T#1S);

IF Pulse.Q THEN
	
	IF Device.Q2 AND tPos>0 THEN tPos:=tPos-1; END_IF;
	IF Device.Q1 AND tPos<100 THEN tPos:=tpos+1; END_IF;
END_IF;


FWD_Limit:=tPos<100;
Rev_Limit:=tPos>0;

END_FUNCTION_BLOCK

// 20 Program Organization Units/Simulators/Eaton_DM1_Sim
FUNCTION Eaton_DM1_Sim : ARRAY[0..10] OF WORD;
VAR_INPUT
	TX:ARRAY[0..10] OF WORD;
END_VAR
VAR
END_VAR

//Status_Word RX[0]
Eaton_DM1_Sim[0].0:=TRUE;	//VFD.Data.Drive_STATUS.Ready:=
Eaton_DM1_Sim[0].1:=TX[0].0;		//VFD.Data.Drive_STATUS.Run:=
Eaton_DM1_Sim[0].2:=TX[0].1;	//VFD.Data.Drive_STATUS.FWD:=



//General Status RX[1]

//Actual Speed RX[2]
IF TX[0].0 THEN
	Eaton_DM1_Sim[2]:=TX[2];	//VFD.Output_Pct:=
	Eaton_DM1_Sim[3]:=(TX[2]/6);		//vfd.Output_Hz:=TO_REAL(
ELSE
	Eaton_DM1_Sim[2]:=0;
	Eaton_DM1_Sim[3]:=0;
END_IF;

Eaton_DM1_Sim[9]:=6240;	//VFD.Data.DC_Link:=TO_REAL(

END_FUNCTION

// 20 Program Organization Units/Simulators/eDip_8412_Sim
FUNCTION eDip_8412_Sim : Bool
VAR_INPUT
	Current:REAL;
	Low_Limit:REAL;
	High_Limit:REAL;
	Rate_Up:REAL;
	Rate_Down:REAL;
END_VAR
VAR
	Data:Bytes_Dword;
END_VAR

VAR_OUTPUT
	RX_0:WORD;
	RX_1:WORD;
END_VAR

Data.tReal:=Current+(Rate_up-Rate_Down);
Data.tReal:=LIMIT(Low_limit,Data.tReal,High_Limit);

RX_0:=Data.tWord[1];
RX_1:=Data.tWord[0];

END_FUNCTION

// 20 Program Organization Units/Simulators/Edip_8691_Sim
FUNCTION Edip_8691_Sim
VAR_INPUT
	BCV: Reference to ceDip_8691;;
END_VAR
VAR_OUTPUT
END_VAR
VAR
END_VAR

//BCV.PDO.EndPositions.0:=BCV.PDO.Setpoint.0;
//BCV.PDO.EndPositions.1:=NOT(BCV.PDO.Setpoint.0);
//BCV.PDO.NamurStatus:=1;


(*
Join.tWord[0]:=BCV.RX[0];
BCV.PDO.EndPositions:=Join.tByte[1];

Join.tWord[0]:=BCV.RX[1];
BCV.PDO.NamurStatus:=Join.tByte[1];
Join.tWord[1]:=BCV.RX[2];
Join.tWord[0]:=BCV.RX[3];
BCV.PDO.Position:=Join.tReal;

Join.tByte[0]:=0;
Join.tByte[1]:=BCV.PDO.Setpoint;
BCV.TX:=Join.tWord[0];
*)

//BCV.RX[0].8:=BCV.TX.8;
//BCV.RX[0].9:=NOT(BCV.TX.8);
//BCV.RX[1]:=256;

END_FUNCTION

// 20 Program Organization Units/Simulators/Edip_8694_Data_Sim
FUNCTION Edip_8694_Data_Sim
VAR_INPUT
END_VAR
VAR_OUTPUT
END_VAR
VAR
	//Data:Bytes_Dword;
END_VAR
VAR_IN_OUT
	Device:ceDip_8694;
END_VAR


Device.RX.ActualPosition.tWord[0]:=Device.TX_CmdDigital.tWord[0];
Device.RX.ActualPosition.tWord[1]:=Device.TX_CmdDigital.tWord[1];

Device.RX.NamurStatus.tByte[1]:=1;

Device.RX.CurrentSetPoint.tWord[0]:=Device.TX_CmdDigital.tWord[0];
Device.RX.CurrentSetPoint.tWord[1]:=Device.TX_CmdDigital.tWord[1];


//Device.RX[5]:=0;

END_FUNCTION

// 20 Program Organization Units/Simulators/eDip_ME44_DI_Count_Sim
FUNCTION eDip_ME44_DI_Count_Sim : Bool
VAR_INPUT
	Pulse_250:BOOL;
	Rate_LPM:REAL;
	FIT:cFIT;
	//Current:REAL;
	
END_VAR
VAR
	//Data:Bytes_Dword;
END_VAR

VAR_OUTPUT
	Count:REAL;
END_VAR



IF NOT(FIT.PLC_Reset) AND NOT(FIT.HMI_Reset) THEN
	IF Pulse_250 THEN
		Count:=TO_REAL(FIT.Counts+(((Rate_LPM/60)/4)*FIT.K));
	ELSE
		Count:=TO_REAL(FIT.Counts);
	END_IF;
ELSE
	Count:=0;	
END_IF;

END_FUNCTION

// 20 Program Organization Units/Simulators/eDip_ME44_DI_Hz_Sim
FUNCTION eDip_ME44_DI_Hz_Sim : Bool
VAR_INPUT

	Rate_LPM:REAL;
	FIT:cFIT;
	
END_VAR
VAR
	//Data:Bytes_Dword;
	//Value:REAL;
END_VAR

VAR_OUTPUT
	Hz:Real;
END_VAR

IF NOT(FIT.PLC_Reset) AND NOT(FIT.HMI_Reset) THEN
	Hz:=(Rate_LPM/60)*FIT.K;
ELSE
	Hz:=0;	
END_IF;

END_FUNCTION

// 20 Program Organization Units/Simulators/FIT_Sim
FUNCTION FIT_Sim : UDINT
VAR_INPUT
	FIT: REFERENCE TO cFIT;
	Control:REAL;
	clk:Bool;
	
END_VAR
VAR_OUTPUT
	Hz:REAL;
END_VAR
VAR
	PLC_Time:UDINT;
END_VAR

IF FIT.HMI_Reset OR FIT.PLC_Reset THEN
	FIT.Counts:=0;
END_IF;

IF clk THEN	
	FIT.Counts:=(FIT.Counts + TO_UDINT(Control/4) );
	IF FIT.Counts=0 THEN FIT.Counts:=1; END_IF;
	
	
END_IF;
FIT_Sim:=FIT.Counts;
Hz:=(Control);

END_FUNCTION

// 20 Program Organization Units/Simulators/HTX_Sim
FUNCTION HTX_Sim : Bool
VAR_INPUT
    A_Rate      : REAL;  (* Mass flow rate of side A *)
    A_InletTemp : REAL;  (* Inlet temperature of side A *)
    B_Rate      : REAL;  (* Mass flow rate of side B *)
    B_InletTemp : REAL;  (* Inlet temperature of side B *)
END_VAR
VAR_OUTPUT
    A_OutletTemp : REAL; (* Outlet temperature of side A *)
    B_OutletTemp : REAL; (* Outlet temperature of side B *)
END_VAR
VAR
    Cp : REAL := 4.18;  (* Specific heat capacity (same for both sides) *)
END_VAR


   // A_OutletTemp := ((A_Rate * A_InletTemp) + (B_Rate * B_InletTemp)) / (A_Rate + B_Rate);
   /// B_OutletTemp := A_OutletTemp; 

    HTX_Sim := TRUE;
(*
IF A_Rate>0.1 THEN
		B_OutletTemp:=((A_Rate * A_InletTemp) + (B_Rate * B_InletTemp)) / (A_Rate + B_Rate);
ELSE	
		A_OutletTemp:= LIMIT(0,A_InletTemp-0.01,100);
END_IF;

IF B_Rate>0.1 THEN
	A_OutletTemp := ((A_Rate * A_InletTemp) + (B_Rate * B_InletTemp)) / (A_Rate + B_Rate);
ELSE
	B_OutletTemp:=LIMIT(0,B_InletTemp-0.01,100);
END_IF
*)

IF A_Rate>0.1 AND B_Rate>0.1 THEN
	A_OutletTemp := ((A_Rate * A_InletTemp) + (B_Rate * B_InletTemp)) / (A_Rate + B_Rate);
	B_OutletTemp:=((A_Rate * A_InletTemp) + (B_Rate * B_InletTemp)) / (A_Rate + B_Rate);
ELSE
	A_OutletTemp:= LIMIT(0,A_InletTemp-0.01,100);
	B_OutletTemp:=LIMIT(0,B_InletTemp-0.01,100);
	
END_IF

END_FUNCTION

// 20 Program Organization Units/Simulators/Mix_Sim
FUNCTION Mix_Sim : REAL;
VAR_INPUT
	HW:REAL;
	CW:REAL;
	Temp:REAL;
	RAW_Scale:cAnalog_scale;
END_VAR
VAR
	
END_VAR
VAR_OUTPUT
	Target_Temp:REAL;
END_VAR

	IF HW<>CW then
		Target_temp:=Burkert_OSCAT_BASIC.SCALE_R(
		X:= ((HW-CW)/(HW+CW)), 
		I_LO:= (-1), 
		I_HI:= 1, 
		O_LO:= 0, 
		O_HI:= Temp);
	ELSE
		Target_Temp:=Temp/2;
	END_IF;
	
	Mix_Sim:=Burkert_OSCAT_BASIC.SCALE_R(
	X:= Target_Temp, 
	I_LO:= Raw_Scale.Eu_Min, 
	I_HI:= Raw_Scale.Eu_Max, 
	O_LO:= Raw_Scale.Raw_Min, 
	O_HI:= Raw_Scale.Raw_Max);

END_FUNCTION

// 20 Program Organization Units/Simulators/Mix_TT_Sim
FUNCTION Mix_TT_Sim : Real
VAR_INPUT
	HWT : REAL;    // Hot Water Temperature
    HWF : REAL;    // Hot Water Flow Rate
    CWT : REAL;    // Cold Water Temperature
    CWF : REAL;    // Cold Water Flow Rate
END_VAR
VAR
END_VAR

IF HWF=0 AND CWF=0 THEN
	MIX_TT_Sim:=MidPoint(A:=CWT,B:=HWT);
ELSE
	MIX_TT_Sim:= (HWT * HWF + CWT * CWF) / (HWF + CWF);
END_IF

END_FUNCTION

// 20 Program Organization Units/Simulators/PipePressure
FUNCTION PipePressure : REAL
VAR_INPUT
    InletPressure : REAL;      // Pressure at the inlet 
    InletFlow     : REAL;      // Flow rate at the inlet 
    OutletFlow    : REAL;      // Flow rate at the outlet 
    StaticLoss    : REAL;      // Static pressure loss 
	K			  :	REAL;		//Flow Error Scaling Factor
END_VAR

VAR_OUTPUT
    DynamicLoss : REAL;
    PressureDrop : REAL;
END_VAR




IF InletFlow>OutletFlow THEN
	DynamicLoss := (InletFlow-OutletFlow) * K; 
	PressureDrop := StaticLoss-DynamicLoss;
END_IF;
IF InletFlow<OutletFlow  THEN
	DynamicLoss := (OutletFlow-InletFlow) * K; 
	PressureDrop := DynamicLoss + StaticLoss;
END_IF;

PipePressure := LIMIT(0,(InletPressure - PressureDrop),InletPressure);

END_FUNCTION

// 20 Program Organization Units/Simulators/SSR_Heater_Sim
FUNCTION SSR_Heater_Sim : REAL;
VAR_INPUT
    HeaterPowerKW     : REAL;  (* Power of the heater in kilowatts (kW) *)
    InletTemp         : REAL;  (* Inlet temperature of the water in degrees Celsius (°C) *)
    InletFlowRateLm   : REAL;  (* Inlet flow rate of the water in liters per minute (L/min) *)
END_VAR
VAR_OUTPUT
	DeltaT:REAL;
END_VAR
VAR
    Cp                : REAL := 4180.0;  (* Specific heat capacity of water in J/kg°C *)
    Rho               : REAL := 1000.0;  (* Density of water in kg/m³ *)
    HeaterPowerW      : REAL;
    FlowRateM3s       : REAL;
    MassFlowRateKgs   : REAL;
    OutletTemp        : REAL;
END_VAR



IF InletFlowRateLm>0  THEN
    HeaterPowerW := HeaterPowerKW * 1000.0;
	FlowRateM3s := (InletFlowRateLm / 1000.0) / 60.0;
	MassFlowRateKgs := Rho * FlowRateM3s;
	DeltaT:=(HeaterPowerW / (MassFlowRateKgs * Cp));
	OutletTemp := DeltaT + InletTemp;
	SSR_Heater_Sim := OutletTemp;
ELSE
	SSR_Heater_Sim:=LIMIT(0,InletTemp,100);
END_IF;

END_FUNCTION

// 20 Program Organization Units/Simulators/Tank_Sim
FUNCTION Tank_Sim : REAL
VAR_INPUT
    Volume            : REAL;  (* Volume of the tank *)
    CurrentTemp       : REAL;  (* Current temperature of the tank *)
    ReturnTemp        : REAL;  (* Temperature of the returning fluid *)
    ReturnRate        : REAL;  (* Flow rate of the returning fluid *)
	TankLoss_Rate		:REAL;
	Trigger				:BOOL; (*500 ms clk*)
END_VAR

VAR_OUTPUT
	TankEnergy      : REAL;
	ReturnVolume	: REAL;
	ReturnEnergy	: REAL;
	TankTempChange	:REAL;
END_VAR
VAR
    Cp                : REAL := 4.18;  (* Specific heat capacity (assumed constant for simplification) *)
    //FinalTemp         : REAL;
    //TotalHeatCapacity : REAL;
    //ReturnHeat        : REAL;
    
END_VAR

ReturnVolume:= ReturnRate/(60*2); (* Rate should always be / Min, Trigger is 500ms so 120 triggers per volume *)
TankEnergy := Volume * Cp * CurrentTemp;
ReturnEnergy := ReturnVolume * Cp * (ReturnTemp-CurrentTemp);
IF Volume>1 THEN
	TankTempChange := ((ReturnEnergy) / (Volume * CP)-TankLoss_Rate);
ELSE
	TankTempChange:=0;
END_IF

IF Trigger THEN
	//FinalTemp := (TankEnergy + ReturnEnergy) / (Volume * CP);
	Tank_Sim := CurrentTemp+TankTempChange;
ELSE
	Tank_Sim:= CurrentTemp;
END_IF

END_FUNCTION

// 20 Program Organization Units/Simulators/TankCND
FUNCTION TankCND : Real
VAR_INPUT
    TankVolume          : REAL;  (* Volume of the tank in liters *)
    InitialConductivity : REAL;  (* Initial conductivity of the tank water in µS/cm *)
    BrineFlowRate       : REAL;  (* Flow rate of the brine solution in liters per minute *)
    BrineConductivity   : REAL;  (* Conductivity of the brine solution in µS/cm *)
    Pulse_1s			:BOOL;
END_VAR
VAR
    TotalBrineVolume   : REAL;
    NewConductivity    : REAL;
END_VAR

TotalBrineVolume := BrineFlowRate /60;
IF Pulse_1s AND TotalBrineVolume>0	THEN
	
	NewConductivity := ((InitialConductivity * TankVolume) + (BrineConductivity * TotalBrineVolume)) / (TankVolume + TotalBrineVolume);
	TankCND:=NewConductivity;
ELSE
	TankCND:=InitialConductivity;
END_IF;

END_FUNCTION

// 20 Program Organization Units/Simulators/TT_SIM
FUNCTION TT_SIM : Bool
VAR_INPUT
	TT: REFERENCE TO cAIT;
	Rate_Up:REAL;
	Rate_Down:REAL;
END_VAR
VAR
END_VAR

TT.Analog_Scale.Raw:=TT.Analog_Scale.Raw+(Rate_up-Rate_Down);
TT.Analog_Scale.Raw:=LIMIT(TT.Analog_Scale.Raw_Min,TT.Analog_Scale.Raw,TT.Analog_Scale.Raw_Max);

END_FUNCTION

// 20 Program Organization Units/Simulators/Vacon_VFD_SIM
FUNCTION_BLOCK Vacon_VFD_SIM
VAR_INPUT
	Device:VFD_Vacon_DUT;
END_VAR
VAR_OUTPUT
END_VAR
VAR
	//Random:REAL;
END_VAR
VAR_IN_OUT
	mbTCP:Vacon_MbTCP;
END_VAR

//Random:=Burkert_OSCAT_BASIC.RDM(Random);
mbTCP.RX[9]:=691;
mbTCP.rx[0].1:=FALSE;// Running Bit
mbTCP.rx[0].2:=TRUE;//FWD BIT;
CASE Device.MODE.eMode	 OF
		VFD_modes.Auto:	IF Device.PLC_Run THEN
					mbTCP.RX[0]:=35;
					mbTCP.rx[0].1:=TRUE;
					mbTCP.rx[0].2:=(Device.PLC_CMD>0);
					mbTCP.RX[3]:=REAL_TO_WORD(ABS(Device.PLC_CMD)*6);
				ELSE
					mbTCP.RX[0]:=1;
					mbTCP.RX[3]:=0;
				END_IF;
		VFD_modes.Disabled:	mbTCP.RX[0]:=1;
			mbTCP.RX[3]:=0;
		VFD_modes.Manual:	mbTCP.RX[0]:=35;
			mbTCP.rx[0].1:=TRUE;
			mbTCP.rx[0].2:=(Device.PLC_CMD>0);
			mbTCP.RX[3]:=REAL_TO_WORD(ABS(Device.MAN_CMD) *6);
END_CASE

END_FUNCTION_BLOCK

// 20 Program Organization Units/Simulators/VFD_GS2x_Sim
FUNCTION VFD_GS2x_Sim : ARRAY[0..11] OF WORD;
VAR_INPUT
	TX:ARRAY[0..2] OF WORD;
END_VAR
VAR
END_VAR

//Status_Word RX[0]
VFD_GS2x_Sim[1].1:=TRUE;	//Status2.1 Ready
VFD_GS2x_Sim[0]:=1;

IF TX[0].1 THEN
	VFD_GS2x_Sim[1].0:=TRUE;		//Run Status2.0
	VFD_GS2x_Sim[3]:=TX[1]/6;			
	//VFD_GS2x_Sim[3]:=(TX[2]/6);		
ELSE
	VFD_GS2x_Sim[1].0:=FALSE;
	VFD_GS2x_Sim[2]:=0;
	//VFD_GS2x_Sim[3]:=0;
END_IF;

VFD_GS2x_Sim[5]:=3610;	//VFD.Data.DC_Link:=TO_REAL(

END_FUNCTION

// 20 Program Organization Units/Simulators/Volume_Sim
FUNCTION_BLOCK Volume_Sim
VAR_INPUT
	Rate_In:REAL;
	Rate_out:REAL;
	Reset:BOOL;
END_VAR
VAR_IN_OUT
	Total:REAL;
END_VAR
VAR
	pulse: Burkert_OSCAT_BASIC.CLK_PRG;
END_VAR

pulse(PT:=T#1S);

IF Pulse.Q THEN
		Total:=Total+(Rate_IN/60.0);
		Total:=Total-(Rate_Out/60.0);
		
END_IF;

IF Reset  OR (Total<0) THEN
	Total:=0;
END_IF;

END_FUNCTION_BLOCK

// 50 Functions/Asi/AC2916
FUNCTION_BLOCK AC2916
VAR_INPUT
	CH1:Asi_node_DUT;
	CH2:ASI_Node_DUT;
END_VAR
VAR_OUTPUT
	AC2916:AC2916_DUT;
END_VAR
VAR
END_VAR

AC2916.AI[1] := Ch1.Analog_RX_0;
AC2916.AI[2] := Ch1.Analog_RX_1;
AC2916.AI[3] := Ch2.Analog_RX_0;
AC2916.AI[4] := Ch2.Analog_RX_1;
AC2916.Active := CH1.Active;
Ac2916.Detected := CH1.Detected;
AC2916.PROJECTED := CH1.PROJECTED;
AC2916.Fault := Ch1.Fault;

END_FUNCTION_BLOCK

// 50 Functions/Asi/Asi_GW_FUN
FUNCTION_BLOCK Asi_GW_FUN
VAR_INPUT
	Flags:ARRAY[0..7] OF DWORD;
	Analog_1_RX:ARRAY[0..79] OF WORD;
	Analog_2_RX:ARRAY[0..74] OF WORD;
	Digital_RX:ARRAY[0..63] OF BYTE;
	
END_VAR
VAR_OUTPUT
	Analog_1_TX:ARRAY[0..79] OF WORD;
	Analog_2_TX:ARRAY[0..74] OF WORD;
	Digital_TX:ARRAY[0..63] OF BYTE;
END_VAR
VAR
	index:INT:=0;
	Offset:INT;
END_VAR

VAR_IN_OUT
	A_Nodes:ARRAY[1..32] OF Asi_node_DUT;
	B_Nodes:ARRAY[1..32] OF Asi_Node_Dut;
END_VAR

FOR index:=1 TO 32 BY 1 DO
	
	A_Nodes[Index].Active:=GETBIT(X:=flags[0] , N:=TO_BYTE(Index) );
	B_Nodes[Index].Active:=GETBIT(X:=flags[1] , N:=TO_BYTE(Index) );
	
	A_Nodes[Index].Detected:=GETBIT(X:=flags[2] , N:=TO_BYTE(Index) );
	B_Nodes[Index].Detected:=GETBIT(X:=flags[3] , N:=TO_BYTE(Index) );
	
	A_Nodes[Index].Fault:=GETBIT(X:=flags[4] , N:=TO_BYTE(Index) );
	B_Nodes[Index].Fault:=GETBIT(X:=flags[5] , N:=TO_BYTE(Index) );
	
	A_Nodes[Index].PROJECTED:=GETBIT(X:=flags[6] , N:=TO_BYTE(Index) );
	B_Nodes[Index].PROJECTED:=GETBIT(X:=flags[7] , N:=TO_BYTE(Index) );
	

	A_Nodes[Index].Digital_RX:=Digital_RX[(Index-1)];
	B_Nodes[Index].Digital_RX:=Digital_RX[(Index+31)];
	
	Digital_TX[Index-1]:=A_Nodes[Index].Digital_TX;
	Digital_TX[Index+31]:=B_Nodes[Index].Digital_TX;
	
	
	IF Index < 17 THEN
		Offset := ((Index-1)*5);
		A_Nodes[Index].Analog_RX_0:=Analog_1_RX[Offset];
		A_Nodes[Index].Analog_RX_1:=Analog_1_RX[Offset+1];
		B_Nodes[Index].Analog_RX_0:=Analog_1_RX[Offset+2];
		B_Nodes[Index].Analog_RX_1:=Analog_1_RX[Offset+3];
		
		Analog_1_TX[Offset]:=A_Nodes[Index].Analog_TX_0;
		Analog_1_TX[Offset+1]:=A_Nodes[Index].Analog_TX_1;
		Analog_1_TX[Offset+2]:=B_Nodes[Index].Analog_TX_0;
		Analog_1_TX[Offset+3]:=B_Nodes[Index].Analog_TX_1;
		
		
	ELSE
		Offset := ((Index-17)*5);
		A_Nodes[Index].Analog_RX_0:=Analog_2_RX[Offset];
		A_Nodes[Index].Analog_RX_1:=Analog_2_RX[Offset+1];
		B_Nodes[Index].Analog_RX_0:=Analog_2_RX[Offset+2];
		B_Nodes[Index].Analog_RX_1:=Analog_2_RX[Offset+3];
		
		Analog_2_TX[Offset]:=A_Nodes[Index].Analog_TX_0;
		Analog_2_TX[Offset+1]:=A_Nodes[Index].Analog_TX_1;
		Analog_2_TX[Offset+2]:=B_Nodes[Index].Analog_TX_0;
		Analog_2_TX[Offset+3]:=B_Nodes[Index].Analog_TX_1;
		
	END_IF;
	
	
END_FOR;

END_FUNCTION_BLOCK

// 50 Functions/Calculators/Calc_SaltPumpSpeed
FUNCTION Calc_SaltPumpSpeed : REAL
VAR_INPUT
    Q_RO 		: REAL;		(* RO Line Flow Rate in GPM *)
    C_target 	: REAL;		(* Target Conductivity in µS/cm *)
    C_salt_PPM 		: REAL:=200_000;     (* Salt Tank Conductivity in µS/cm *)
    Q_salt_max 	: REAL;  	(* Max Salt Pump Flow Rate in GPM *)
END_VAR

VAR_OUTPUT
	 Q_salt : REAL;      	(* Required Salt Flow Rate in GPM *)
END_VAR


VAR
	C_target_ppm 	: REAL; 	(*target concentration in ppm*)
	//C_salt_ppm 		: REAL;		(*salt tank concentration in ppm*)
END_VAR

C_target_ppm:= 0.4195*C_target - 5.2485; (*Note IF value negative, set TO 0*)
//C_salt_ppm:=200000;	(* <unknown>, set TO 200,000 ppm (we will need curve FOR THIS some TIME FROM BASF presumably)   *)


 IF  C_salt_ppm >C_target_ppm THEN
        //Q_salt := (C_target * Q_RO) / (C_salt - C_target);
		Q_salt := (C_target_ppm * Q_RO) / (C_salt_ppm - C_target_ppm);
    ELSE
        Q_salt := 0; (* If salt conductivity is too low, do not inject *)
    END_IF;

    (* Calculate Pump Speed as a Percentage of Max Flow *)
    IF Q_salt_max > 0 THEN
        Calc_SaltPumpSpeed := (Q_salt / Q_salt_max) * 100;
    ELSE
        Calc_SaltPumpSpeed := 0; (* Avoid division by zero *)
    END_IF;

END_FUNCTION

// 50 Functions/Calculators/Calculate_Chlorine_Volume
FUNCTION Calculate_Chlorine_Volume : REAL
VAR_INPUT
	Target_PPM : REAL;  (* Desired PPM in the destination vessel *)
    Water_Volume_USG : REAL;  (* Volume of water in US Gallons *)
    Source_Concentration : REAL;  (* Source chlorine concentration as a decimal (e.g., 40% = 0.40) *)
END_VAR


VAR	
	Water_Volume_L : REAL;
    Chlorine_Mass_mg : REAL;
    Chlorine_Volume_L : REAL;
    Chlorine_Volume_USG : REAL;
END_VAR

IF Source_Concentration>0 THEN

	(* Convert water volume from US Gallons to Liters *)
	Water_Volume_L := Water_Volume_USG * 3.785;
	
	(* Calculate required mass of chlorine in mg *)
	Chlorine_Mass_mg := Target_PPM * Water_Volume_L;
	
	(* Calculate required volume of chlorine solution in Liters *)
	Chlorine_Volume_L := Chlorine_Mass_mg / ((Source_Concentration/100) * 1_000_000);
	
	(* Convert Chlorine volume to US Gallons *)
	Chlorine_Volume_USG := Chlorine_Volume_L / 3.785;
	
	(* Return the required volume in US Gallons *)
	Calculate_Chlorine_Volume := Chlorine_Volume_USG;
ELSE
	Calculate_Chlorine_Volume:=0;
END_IF

END_FUNCTION

// 50 Functions/Calculators/DilutionOutput
FUNCTION DilutionOutput : Bool
VAR_INPUT
    A_Rate : REAL;     // Flow rate of Stream A (LPM)
    A_Strength : REAL; // Strength of Stream A (% or any concentration unit)
    B_Rate : REAL;     // Flow rate of Stream B (LPM)
    B_Strength : REAL; // Strength of Stream B (% or any concentration unit)
END_VAR
VAR_OUTPUT
    C_Rate : REAL;     // Combined flow rate (LPM)
    C_Strength : REAL; // Combined concentration (% or any concentration unit)
END_VAR

// Calculate combined flow rate
C_Rate := A_Rate + B_Rate;

// Calculate combined concentration if flow rate is greater than 0
IF C_Rate > 0 THEN
    C_Strength := (A_Rate * A_Strength + B_Rate * B_Strength) / C_Rate;
ELSE
    C_Strength := 0;
END_IF;

// Indicate successful calculation
DilutionOutput := TRUE;

END_FUNCTION

// 50 Functions/Calculators/KV_Calculator
FUNCTION KV_Calculator : Real
VAR_INPUT
	FR : REAL;            // Flow rate in LPM
    DeltaP : REAL;       // Pressure drop in psi
    SG : REAL;           // Specific gravity of the fluid
END_VAR
VAR
END_VAR

IF DeltaP>0 AND FR>0 AND SG>0 THEN
	KV_Calculator:= ((FR*0.06) * SQRT(SG / (DeltaP * 0.0705)));
ELSE
	KV_Calculator:=0.0;
END_IF;

END_FUNCTION

// 50 Functions/Calculators/VolumeBasedDilution
FUNCTION VolumeBasedDilution : Bool
VAR_INPUT
    A_Volume : REAL;     // Volume of Stream A
    A_Strength : REAL;   // Strength of Stream A (% or any concentration unit)
    B_Volume : REAL;     // Volume of Stream B
    B_Strength : REAL;   // Strength of Stream B (% or any concentration unit)
END_VAR
VAR_OUTPUT
    C_Volume : REAL;     // Combined Volume
    C_Strength : REAL;   // Combined Concentration (% or any concentration unit)
END_VAR

// Calculate combined volume
C_Volume := A_Volume + B_Volume;

// Calculate combined concentration if volume is greater than 0
IF C_Volume > 0 THEN
    C_Strength := (A_Volume * A_Strength + B_Volume * B_Strength) / C_Volume;
ELSE
    C_Strength := 0;
END_IF;

// Indicate successful calculation
VolumeBasedDilution := TRUE;

END_FUNCTION

// 50 Functions/NVL/f_Fermenter_To_NVL
FUNCTION f_Fermenter_To_NVL : Bool
VAR_INPUT
	LCL:cFermenter_DUT;
END_VAR
VAR_OUTPUT
	NVL:cFermenter_NVL;
END_VAR
VAR
END_VAR

NVL.Crash_Target:=LCL.Crash_Target;

END_FUNCTION

// 20 Program Organization Units/HMI_Sync/Level_0/HMI_8228_Sync
FUNCTION HMI_8228_Sync : Bool
VAR_INPUT
	//EN:BOOL;

END_VAR
VAR
	//r_trig_0:r_trig;
END_VAR

VAR_IN_OUT;
	Local:c8228;
	HMI:c8228;
END_VAR


local.Locate:=HMI.Locate;
Local.Maintenance:=HMI.Maintenance;	
HMI:=Local;

END_FUNCTION

// 20 Program Organization Units/HMI_Sync/Level_0/HMI_8605_Sync
FUNCTION_BLOCK HMI_8605_Sync
VAR_INPUT
	Sync:BOOL;
	HMI:REFERENCE TO c8605;
	Local:REFERENCE TO c8605;
END_VAR
VAR_OUTPUT
	strNamur:String[30];
END_VAR
VAR
	Buffer_locate:BOOL;
	Buffer_ReadOnce:BOOL;
	Sync_Trig:R_Trig;
	Valid:Bool;
END_VAR

Valid:= __ISVALIDREF(HMI) AND __ISVALIDREF(Local);
IF Valid THEN
	
	Sync_Trig(CLK:=Sync);
	IF Sync_trig.Q THEN
		HMI:=Local;
		Buffer_Locate:=Local.Locate;
	END_IF;
	IF Sync THEN
		IF HMI.Locate=Buffer_locate  THEN
			HMI:=Local;
		ELSE
			local.Locate:=				HMI.Locate;
			Buffer_Locate:=HMI.Locate;
			HMI:=Local;
		END_IF
	END_IF;
	
END_IF



//strMode:=Burkert_OSCAT_BASIC.REPLACE_ALL(str:=TO_STRING(local.Mode.eMode), src:='_' , rep:=' ' );
//strStatus:=Burkert_OSCAT_BASIC.REPLACE_ALL(str:=TO_STRING(local.Status.eStatus), src:='_' , rep:=' ' );
strNamur:=Burkert_OSCAT_BASIC.REPLACE_ALL(str:=TO_STRING(Local.PDO.Namur.eNamur), src:='_' , rep:=' ' );

END_FUNCTION_BLOCK

// 20 Program Organization Units/HMI_Sync/Level_0/HMI_8653_Sync
FUNCTION HMI_8653_Sync : Bool
VAR_INPUT
	//EN:BOOL;

END_VAR
VAR
	//r_trig_0:r_trig;
END_VAR

VAR_IN_OUT;
	Local:c8653;
	HMI:c8653;
END_VAR


local.Locate:=HMI.Locate;
Local.Maintenance:=HMI.Maintenance;
Local.SDO.Counter_Reset:=Local.SDO.Counter_Reset;	
HMI:=Local;

END_FUNCTION

// 20 Program Organization Units/HMI_Sync/Level_0/HMI_ME44AI_Sync
FUNCTION HMI_ME44AI_Sync : Bool
VAR_INPUT
	//EN:BOOL;

END_VAR
VAR
	//r_trig_0:r_trig;
END_VAR

VAR_IN_OUT;
	Local:cME44_AI;
	HMI:cME44_AI;
END_VAR


local.Locate:=HMI.Locate;
Local.Maintenance:=HMI.Maintenance;	
HMI:=Local;

END_FUNCTION

// 20 Program Organization Units/HMI_Sync/Level_0/HMI_ME64_Sync
FUNCTION HMI_ME64_Sync : Bool
VAR_INPUT
	//EN:BOOL;

END_VAR
VAR
	//r_trig_0:r_trig;
END_VAR

VAR_IN_OUT;
	Local:cME64;
	HMI:cME64;
END_VAR


local.Locate:=HMI.Locate;
Local.Maintenance:=HMI.Maintenance;	
HMI:=Local;

END_FUNCTION

// 20 Program Organization Units/HMI_Sync/Level_1/ACV_HMI_Sync_UDFB
FUNCTION_BLOCK ACV_HMI_Sync_UDFB
VAR_INPUT
	Sync:BOOL;
END_VAR
VAR_OUTPUT
	strMode:STRING;
	strStatus:STRING;
END_VAR
VAR
	Buffer:cACV;
	R_Trig_0: R_trig;
	Sync_1: BOOL;
	Sync_2: BOOL;
	PLC_Changes:UINT;
	HMI_Changes:UINT;
	
	HMI_Change: BOOL;
END_VAR

VAR_IN_OUT
	HMI:cACV;
	Local:cACV;
END_VAR

(* body of a kind this reader does not render *)

END_FUNCTION_BLOCK

// 20 Program Organization Units/HMI_Sync/Level_1/AIT_HMI_Sync_UDFB
FUNCTION_BLOCK AIT_HMI_Sync_UDFB
VAR_INPUT
	Sync:BOOL;
END_VAR
VAR_OUTPUT
	strMode:STRING;
	strStatus:STRING;
END_VAR
VAR
	Buffer:cAIT;
	R_Trig_0: R_trig;
	Sync_1: BOOL;
	Sync_2: BOOL;
	PLC_Changes:UINT;
	HMI_Changes:UINT;
	
	Clear_F_Trig: F_trig;
END_VAR

VAR_IN_OUT
	HMI:cAIT;
	Local:cAIT;
END_VAR

(* body of a kind this reader does not render *)

END_FUNCTION_BLOCK

// 20 Program Organization Units/HMI_Sync/Level_1/B8050_HMI_Sync_UDFB
FUNCTION_BLOCK B8050_HMI_Sync_UDFB
VAR_INPUT
	//Sync:BOOL;
	Index:UINT;
	Max_Index:UINT;
END_VAR
VAR_OUTPUT
END_VAR
VAR
	R_Trig_0: R_trig;
	//Buffer_HMI_reset:BOOL;
	Sync:BOOL;
END_VAR

VAR_IN_OUT
	//HMI:c8050;
	//Local:c8050;
END_VAR

(* body of a kind this reader does not render *)

END_FUNCTION_BLOCK

// 20 Program Organization Units/HMI_Sync/Level_1/BCV_HMI_Sync_UDFB
FUNCTION_BLOCK BCV_HMI_Sync_UDFB
VAR_INPUT
	Sync:BOOL;
END_VAR
VAR_OUTPUT
	strMode:STRING;
	strStatus:STRING;
END_VAR
VAR
	Buffer:cBCV;
	R_Trig_0: R_trig;
	Sync_1: BOOL;
	Sync_2: BOOL;
	PLC_Changes:UINT;
	HMI_Changes:UINT;
	
END_VAR

VAR_IN_OUT
	HMI:cBCV;
	Local:cBCV;
END_VAR

(* body of a kind this reader does not render *)

END_FUNCTION_BLOCK

// 20 Program Organization Units/HMI_Sync/Level_1/c8691_HMI_Sync_UDFB
FUNCTION_BLOCK c8691_HMI_Sync_UDFB
VAR_INPUT
	Sync:BOOL;
END_VAR
VAR_OUTPUT
	strMode:STRING;
	strStatus:STRING;
END_VAR
VAR
	Buffer:cDigital_BCV;
	R_Trig_0: R_trig;
	Sync_1: BOOL;
	Sync_2: BOOL;
	PLC_Changes:UINT;
	HMI_Changes:UINT;
	
END_VAR

VAR_IN_OUT
	HMI:cDigital_BCV;
	Local:cDigital_BCV;
END_VAR

(* body of a kind this reader does not render *)

END_FUNCTION_BLOCK

// 20 Program Organization Units/HMI_Sync/Level_1/c8694_HMI_Sync_UDFB
FUNCTION_BLOCK c8694_HMI_Sync_UDFB
VAR_INPUT
	Sync:BOOL;
END_VAR
VAR_OUTPUT
	strMode:STRING;
	strStatus:STRING;
	StrNamurNe107:STRING;
END_VAR
VAR
	Buffer:cDigital_ACV;
	R_Trig_0: R_trig;
	Sync_1: BOOL;
	Sync_2: BOOL;
	PLC_Changes:UINT;
	HMI_Changes:UINT;
	
	HMI_Change: BOOL;
END_VAR

VAR_IN_OUT
	HMI:cDigital_ACV;
	Local:cDigital_ACV;
END_VAR

(* body of a kind this reader does not render *)

END_FUNCTION_BLOCK

// 20 Program Organization Units/HMI_Sync/Level_1/Contactor_HMI_Sync_UDFB
FUNCTION_BLOCK Contactor_HMI_Sync_UDFB
VAR_INPUT
	Sync:BOOL;
END_VAR
VAR_OUTPUT
	strMode:STRING;
	strStatus:STRING;
END_VAR
VAR
	Buffer:Contactor_DUT;
	R_Trig_0: R_trig;
	Sync_1: BOOL;
	Sync_2: BOOL;
	PLC_Changes:UINT;
	HMI_Changes:UINT;
	
END_VAR

VAR_IN_OUT
	HMI:Contactor_DUT;
	Local:Contactor_DUT;
END_VAR

(* body of a kind this reader does not render *)

END_FUNCTION_BLOCK

// 20 Program Organization Units/HMI_Sync/Level_1/DI_HMI_Sync_UDFB
FUNCTION_BLOCK DI_HMI_Sync_UDFB
VAR_INPUT
	Sync:BOOL;
END_VAR
VAR_OUTPUT
	strMode:STRING;
	strStatus:STRING;
END_VAR
VAR
	Buffer:DI_DUT;
	R_Trig_0: R_trig;
	Sync_1: BOOL;
	Sync_2: BOOL;
	PLC_Changes:UINT;
	HMI_Changes:UINT;
	
END_VAR

VAR_IN_OUT
	HMI:DI_DUT;
	Local:DI_DUT;
END_VAR

(* body of a kind this reader does not render *)

END_FUNCTION_BLOCK

// 20 Program Organization Units/HMI_Sync/Level_1/DO_HMI_Sync_UDFB
FUNCTION_BLOCK DO_HMI_Sync_UDFB
VAR_INPUT
	Sync:BOOL;
END_VAR
VAR_OUTPUT
	strMode:STRING;
	strStatus:STRING;
END_VAR
VAR
	Buffer:DO_DUT;
	R_Trig_0: R_trig;
	Sync_1: BOOL;
	Sync_2: BOOL;
	PLC_Changes:UINT;
	HMI_Changes:UINT;
	
END_VAR

VAR_IN_OUT
	HMI:DO_DUT;
	Local:DO_DUT;
END_VAR

(* body of a kind this reader does not render *)

END_FUNCTION_BLOCK

// 20 Program Organization Units/HMI_Sync/Level_1/eDip_s8228_HMI_Sync
FUNCTION_BLOCK eDip_s8228_HMI_Sync
VAR_INPUT
	Sync:BOOL;
END_VAR
VAR_OUTPUT
	strMode:STRING;
	strStatus:STRING;
	
	StrConcentration	:STRING;
	StrConductivity		:STRING;
	StrResistivity		:STRING;
	StrTDS				:STRING;
	STRTemperature		:STRING;
	
END_VAR
VAR
	Buffer:c8228;
	R_Trig_0: R_trig;
	Sync_1: BOOL;
	Sync_2: BOOL;
	PLC_Changes:UINT;
	HMI_Changes:UINT;
	
END_VAR

VAR_IN_OUT
	HMI:c8228;
	Local:c8228;
END_VAR

(* body of a kind this reader does not render *)

END_FUNCTION_BLOCK

// 20 Program Organization Units/HMI_Sync/Level_1/FB_HMIAlarmBinder
FUNCTION_BLOCK FB_HMIAlarmBinder
VAR_INPUT
  
	//HMI_cAlarm : REFERENCE TO cAlarm_Config;
END_VAR
VAR_OUTPUT
    Bound       : BOOL;
END_VAR

IF NOT(__ISVALIDREF(HMI.Ref_cAlarm)) THEN UnBind(); END_IF;

END_FUNCTION_BLOCK

// 20 Program Organization Units/HMI_Sync/Level_1/FIT_HMI_Sync_UDFB
FUNCTION_BLOCK FIT_HMI_Sync_UDFB
VAR_INPUT
	Sync:BOOL;
END_VAR
VAR_OUTPUT
	strMode:STRING;
	StrStatus:STRING;
END_VAR
VAR
	Buffer:cFIT;
	R_Trig_0: R_trig;
	Sync_1: BOOL;
	Sync_2: BOOL;
	PLC_Changes:UINT;
	HMI_Changes:UINT;
	
END_VAR

VAR_IN_OUT
	HMI:cFIT;
	Local:cFIT;
END_VAR

(* body of a kind this reader does not render *)

END_FUNCTION_BLOCK

// 20 Program Organization Units/HMI_Sync/Level_1/s336x_HMI_Sync
FUNCTION_BLOCK s336x_HMI_Sync
VAR_INPUT
	Sync:BOOL;
END_VAR
VAR_OUTPUT
	strMode:STRING;
	strStatus:STRING;
	StrNamurNe107:STRING;
END_VAR
VAR
	Buffer:c336x;
	R_Trig_0: R_trig;
	Sync_1: BOOL;
	Sync_2: BOOL;
	PLC_Changes:UINT;
	HMI_Changes:UINT;
	
	HMI_Change: BOOL;
END_VAR

VAR_IN_OUT
	HMI:c336x;
	Local:c336x;
END_VAR

(* body of a kind this reader does not render *)

END_FUNCTION_BLOCK

// 20 Program Organization Units/HMI_Sync/Level_1/s8050_HMI_Sync
FUNCTION_BLOCK s8050_HMI_Sync
VAR_INPUT
	Sync:BOOL;
	Alarm_index:UINT;
	HMIAlarmBinder :REFERENCE TO FB_HMIAlarmBinder;
END_VAR
VAR_OUTPUT
	strMode:STRING;
	strStatus:STRING;
END_VAR
VAR
	Buffer:c8050;
	R_Trig_0: R_trig;
	Sync_1: BOOL;
	Sync_2: BOOL;
	PLC_Changes:UINT;
	HMI_Changes:UINT;
	
	Bind_R_trig: R_Trig;
	UnBind_R_trig: R_Trig;
END_VAR

VAR_IN_OUT
	HMI:c8050;
	Local:c8050;
END_VAR

(* body of a kind this reader does not render *)

END_FUNCTION_BLOCK

// 20 Program Organization Units/HMI_Sync/Level_1/s8098_HMI_Sync_UDFB
FUNCTION_BLOCK s8098_HMI_Sync_UDFB
VAR_INPUT
	Sync:BOOL;
END_VAR
VAR_OUTPUT
	//strMode:STRING;
	strNamur:STRING;
END_VAR
VAR
	Buffer:c8098;
	R_Trig_0: R_trig;
	Sync_1: BOOL;
	Sync_2: BOOL;
	PLC_Changes:UINT;
	HMI_Changes:UINT;
	
END_VAR

VAR_IN_OUT
	HMI:c8098;
	Local:c8098;
END_VAR

VAR_OUTPUT
	//Name:String;
END_VAR

(* body of a kind this reader does not render *)

END_FUNCTION_BLOCK

// 20 Program Organization Units/HMI_Sync/Level_1/s8312_HMI_Sync
FUNCTION_BLOCK s8312_HMI_Sync
VAR_INPUT
	Sync:BOOL;
END_VAR
VAR_OUTPUT
	strMode:STRING;
	strStatus:STRING;
END_VAR
VAR
	Buffer:c8312;
	R_Trig_0: R_trig;
	Sync_1: BOOL;
	Sync_2: BOOL;
	PLC_Changes:UINT;
	HMI_Changes:UINT;
	
END_VAR

VAR_IN_OUT
	HMI:c8312;
	Local:c8312;
END_VAR

(* body of a kind this reader does not render *)

END_FUNCTION_BLOCK

// 20 Program Organization Units/HMI_Sync/Level_1/s8412_HMI_Sync
FUNCTION_BLOCK s8412_HMI_Sync
VAR_INPUT
	Sync:BOOL;
END_VAR
VAR_OUTPUT
	strMode:STRING;
	strStatus:STRING;
END_VAR
VAR
	Buffer:c8412;
	R_Trig_0: R_trig;
	Sync_1: BOOL;
	Sync_2: BOOL;
	PLC_Changes:UINT;
	HMI_Changes:UINT;
	
END_VAR

VAR_IN_OUT
	HMI:c8412;
	Local:c8412;
END_VAR

(* body of a kind this reader does not render *)

END_FUNCTION_BLOCK

// 20 Program Organization Units/HMI_Sync/Level_1/SV_HMI_Sync
FUNCTION_BLOCK SV_HMI_Sync
VAR_INPUT
	Sync:BOOL;
END_VAR
VAR_OUTPUT
	strMode:STRING;
	strStatus:STRING;
END_VAR
VAR
	Buffer:SV_DUT;
	R_Trig_0: R_trig;
	Sync_1: BOOL;
	Sync_2: BOOL;
	PLC_Changes:UINT;
	HMI_Changes:UINT;
	
END_VAR

VAR_IN_OUT
	HMI:SV_DUT;
	Local:SV_DUT;
END_VAR

(* body of a kind this reader does not render *)

END_FUNCTION_BLOCK

// 20 Program Organization Units/HMI_Sync/Level_2/Chase_HMI_Sync_UDFB
FUNCTION_BLOCK Chase_HMI_Sync_UDFB
VAR_INPUT
	Sync:BOOL;
END_VAR
VAR_OUTPUT
END_VAR
VAR
	Buffer:cChase;
	R_Trig_0: R_trig;
	Sync_1: BOOL;
	Sync_2: BOOL;
	PLC_Changes:UINT;
	HMI_Changes:UINT;
	
END_VAR

VAR_IN_OUT
	HMI:cChase;
	Local:cChase;
END_VAR

(* body of a kind this reader does not render *)

END_FUNCTION_BLOCK

// 20 Program Organization Units/HMI_Sync/Level_2/Condensate_HMI_Sync_UDFB
FUNCTION_BLOCK Condensate_HMI_Sync_UDFB
VAR_INPUT
	Sync:BOOL;
END_VAR
VAR_OUTPUT
	StrStatus:STRING;
	StrMode:String;
END_VAR
VAR
	Buffer:cCondensate_Trap;
	R_Trig_0: R_trig;
	Sync_1: BOOL;
	Sync_2: BOOL;
	PLC_Changes:UINT;
	HMI_Changes:UINT;
	
END_VAR

VAR_IN_OUT
	HMI:cCondensate_Trap;
	Local:cCondensate_Trap;
END_VAR

(* body of a kind this reader does not render *)

END_FUNCTION_BLOCK

// 20 Program Organization Units/HMI_Sync/Level_2/PID_HMI_Sync_UDFB
FUNCTION_BLOCK PID_HMI_Sync_UDFB
VAR_INPUT
	Sync:BOOL;
END_VAR
VAR_OUTPUT
	strMode:STRING;
	strStatus:STRING;
END_VAR
VAR
	Buffer:PID_DUT;
	R_Trig_0: R_trig;
	Sync_1: BOOL;
	Sync_2: BOOL;
	PLC_Changes:UINT;
	HMI_Changes:UINT;
	
END_VAR

VAR_IN_OUT
	HMI:PID_DUT;
	Local:PID_DUT;
END_VAR

(* body of a kind this reader does not render *)

END_FUNCTION_BLOCK

// 20 Program Organization Units/HMI_Sync/Level_2/Quick_Mix_HMI_Sync_UDFB
FUNCTION_BLOCK Quick_Mix_HMI_Sync_UDFB
VAR_INPUT
	Sync:BOOL;
END_VAR
VAR_OUTPUT
	//tAIT:AIT_DUT;
END_VAR
VAR
	Buffer:Quick_Mix_DUT;
	R_Trig_0: R_trig;
	Sync_1: BOOL;
	Sync_2: BOOL;
	PLC_Changes:UINT;
	HMI_Changes:UINT;
	
END_VAR

VAR_IN_OUT
	HMI:Quick_mix_DUT;
	Local:Quick_mix_DUT;
END_VAR

VAR_OUTPUT
	strMode:STRING;
	strStatus:STRING;
END_VAR

(* body of a kind this reader does not render *)

END_FUNCTION_BLOCK

// 20 Program Organization Units/HMI_Sync/Level_2/SW_HMI_Sync_UDFB
FUNCTION_BLOCK SW_HMI_Sync_UDFB
VAR_INPUT
	Sync:BOOL;
END_VAR
VAR_OUTPUT
	strMode:STRING;
	strStatus:STRING;
END_VAR
VAR
	Buffer:cBatch_Transfer;
	R_Trig_0: R_trig;
	Sync_1: BOOL;
	Sync_2: BOOL;
	PLC_Changes:UINT;
	HMI_Changes:UINT;
	
END_VAR

VAR_IN_OUT
	HMI:cBatch_Transfer;
	Local:cBatch_Transfer;
END_VAR

(* body of a kind this reader does not render *)

END_FUNCTION_BLOCK

// 20 Program Organization Units/HMI_Sync/Level_3/Brite_HMI_Sync
FUNCTION_BLOCK Brite_HMI_Sync
VAR_INPUT
	Sync:BOOL;
END_VAR
VAR_OUTPUT
END_VAR
VAR
	Buffer:cBrite_DUT;
	R_Trig_0: R_trig;
	Sync_1: BOOL;
	Sync_2: BOOL;
	PLC_Changes:UINT;
	HMI_Changes:UINT;
	
	//PID_0: PID_HMI_Sync_UDFB;
	PID_Match: BOOL;
	Status_Match: BOOL;
	PID_Coompare: UINT;
	Status_Compare: UINT;
END_VAR

VAR_IN_OUT
	HMI:cBrite_DUT;
	Local:cBrite_DUT;
END_VAR

(* body of a kind this reader does not render *)

END_FUNCTION_BLOCK

// 20 Program Organization Units/HMI_Sync/Level_3/Fermenter_HMI_Sync
FUNCTION_BLOCK Fermenter_HMI_Sync
VAR_INPUT
	Sync:BOOL;
END_VAR
VAR_OUTPUT
END_VAR
VAR
	Buffer:cFermenter_DUT;
	R_Trig_0: R_trig;
	Sync_1: BOOL;
	Sync_2: BOOL;
	PLC_Changes:UINT;
	HMI_Changes:UINT;
	
	//PID_0: PID_HMI_Sync_UDFB;
	PID_Match: BOOL;
	Status_Match: BOOL;
	PID_Coompare: UINT;
	Status_Compare: UINT;
END_VAR

VAR_IN_OUT
	HMI:cFermenter_DUT;
	Local:cFermenter_DUT;
END_VAR

(* body of a kind this reader does not render *)

END_FUNCTION_BLOCK

// 20 Program Organization Units/Level_0_Remote_IO/Advantech/Adam_6015_FB
FUNCTION Adam_6015_FB : BOOL
VAR_INPUT
	RX: ARRAY[0..6] OF REAL;
	BurnOut: WORD;
	Comms_Status:WagoSysModbusDiag.eChannelError;
END_VAR
VAR_OUTPUT
	RTD_0:REAL;
	//RTD_0_Fault:BOOL;
	RTD_1:REAL;
	//RTD_1_Fault:BOOL;
	RTD_2:REAL;
	//RTD_2_Fault:BOOL;
	RTD_3:REAL;
	//RTD_3_Fault:BOOL;
	RTD_4:REAL;
	//RTD_4_Fault:BOOL;
	RTD_5:REAL;
	//RTD_5_Fault:BOOL;
	RTD_6:REAL;
	//RTD_6_Fault:BOOL;
END_VAR
VAR
END_VAR

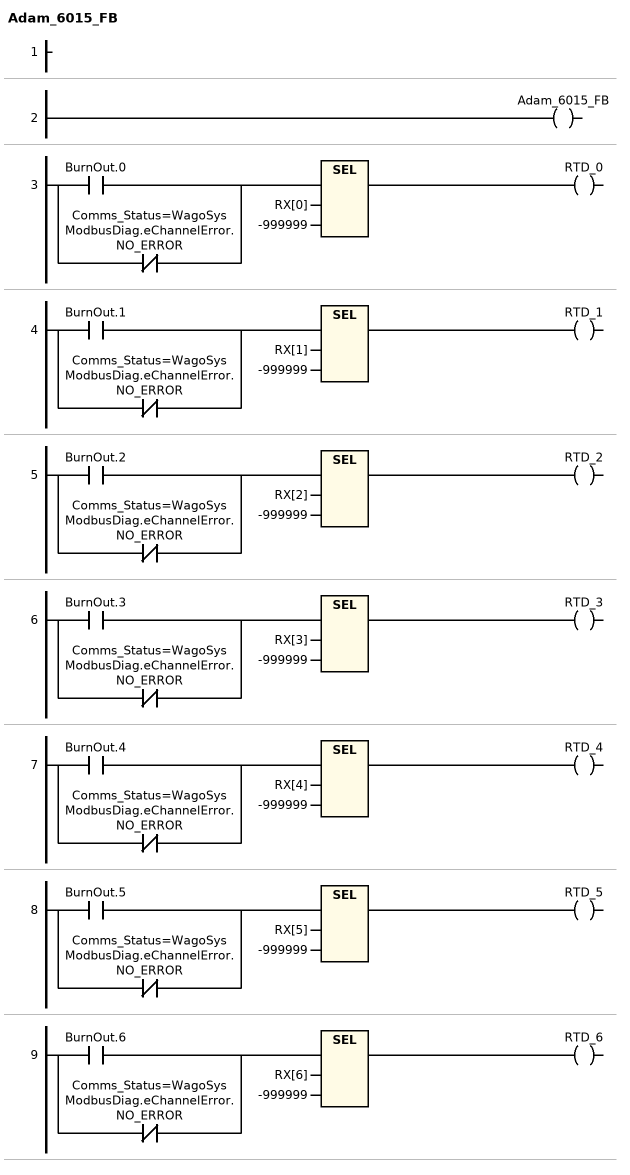
// NETWORK 1

// NETWORK 2
Adam_6015_FB := TRUE;

// NETWORK 3
RTD_0 := SEL(BurnOut.0 OR NOT (Comms_Status=WagoSysModbusDiag.eChannelError.NO_ERROR), RX[0], -999999);

// NETWORK 4
RTD_1 := SEL(BurnOut.1 OR NOT (Comms_Status=WagoSysModbusDiag.eChannelError.NO_ERROR), RX[1], -999999);

// NETWORK 5
RTD_2 := SEL(BurnOut.2 OR NOT (Comms_Status=WagoSysModbusDiag.eChannelError.NO_ERROR), RX[2], -999999);

// NETWORK 6
RTD_3 := SEL(BurnOut.3 OR NOT (Comms_Status=WagoSysModbusDiag.eChannelError.NO_ERROR), RX[3], -999999);

// NETWORK 7
RTD_4 := SEL(BurnOut.4 OR NOT (Comms_Status=WagoSysModbusDiag.eChannelError.NO_ERROR), RX[4], -999999);

// NETWORK 8
RTD_5 := SEL(BurnOut.5 OR NOT (Comms_Status=WagoSysModbusDiag.eChannelError.NO_ERROR), RX[5], -999999);

// NETWORK 9
RTD_6 := SEL(BurnOut.6 OR NOT (Comms_Status=WagoSysModbusDiag.eChannelError.NO_ERROR), RX[6], -999999);

END_FUNCTION

// 20 Program Organization Units/Level_0_Remote_IO/Advantech/Adam_6050_FB
FUNCTION Adam_6050_FB : BOOL
VAR_INPUT
	HSC_0_Enable:BOOL:=FALSE;
	HSC_0_Reset:BOOL:=FALSE;
	HSC_1_Enable:BOOL:=FALSE;
	HSC_1_Reset:BOOL:=FALSE;
	HSC_2_Enable:BOOL:=FALSE;
	HSC_2_Reset:BOOL:=FALSE;
	HSC_3_Enable:BOOL:=FALSE;
	HSC_3_Reset:BOOL:=FALSE;
	HSC_4_Enable:BOOL:=FALSE;
	HSC_4_Reset:BOOL:=FALSE;
	HSC_5_Enable:BOOL:=FALSE;
	HSC_5_Reset:BOOL:=FALSE;
	HSC_6_Enable:BOOL:=FALSE;
	HSC_6_Reset:BOOL:=FALSE;
	HSC_7_Enable:BOOL:=FALSE;
	HSC_7_Reset:BOOL:=FALSE;
	HSC_8_Enable:BOOL:=FALSE;
	HSC_8_Reset:BOOL:=FALSE;
	HSC_9_Enable:BOOL:=FALSE;
	HSC_9_Reset:BOOL:=FALSE;
	HSC_10_Enable:BOOL:=FALSE;
	HSC_10_Reset:BOOL:=FALSE;
	HSC_11_Enable:BOOL:=FALSE;
	HSC_11_Reset:BOOL:=FALSE;
	
	DO_0:BOOL:=FALSE;
	DO_1:BOOL:=FALSE;
	DO_2:BOOL:=FALSE;
	DO_3:BOOL:=FALSE;
	DO_4:BOOL:=FALSE;
	DO_5:BOOL:=FALSE;
//	DO_6:BOOL;
//	DO_7:BOOL;
	RX_DI: WORD;
	RX_Counts: ARRAY[0..11] OF UDINT;
END_VAR
VAR_OUTPUT
	HSC_0:UDINT;
	HSC_1:UDINT;
	HSC_2:UDINT;
	HSC_3:UDINT;
	HSC_4:UDINT;
	HSC_5:UDINT;
	HSC_6:UDINT;
	HSC_7:UDINT;
	HSC_8:UDINT;
	HSC_9:UDINT;
	HSC_10:UDINT;
	HSC_11:UDINT;
	
	DI_0:BOOL;
	DI_1:BOOL;
	DI_2:BOOL;
	DI_3:BOOL;
	DI_4:BOOL;
	DI_5:BOOL;
	DI_6:BOOL;
	DI_7:BOOL;
	DI_8:BOOL;
	DI_9:BOOL;
	DI_10:BOOL;
	DI_11:BOOL;
	
	

	
	
	TX_DO: WORD;
	TX_Counts_Control: ARRAY[0..2] OF WORD;
END_VAR
VAR
END_VAR

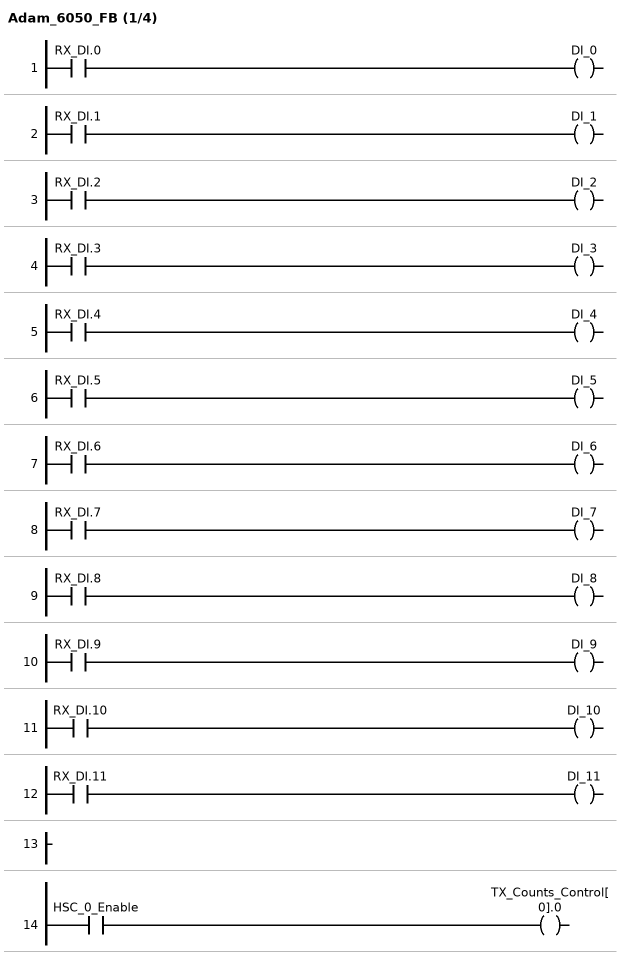
// NETWORK 1
DI_0 := RX_DI.0;

// NETWORK 2
DI_1 := RX_DI.1;

// NETWORK 3
DI_2 := RX_DI.2;

// NETWORK 4
DI_3 := RX_DI.3;

// NETWORK 5
DI_4 := RX_DI.4;

// NETWORK 6
DI_5 := RX_DI.5;

// NETWORK 7
DI_6 := RX_DI.6;

// NETWORK 8
DI_7 := RX_DI.7;

// NETWORK 9
DI_8 := RX_DI.8;

// NETWORK 10
DI_9 := RX_DI.9;

// NETWORK 11
DI_10 := RX_DI.10;

// NETWORK 12
DI_11 := RX_DI.11;

// NETWORK 13

// NETWORK 14
TX_Counts_Control[0].0 := HSC_0_Enable;

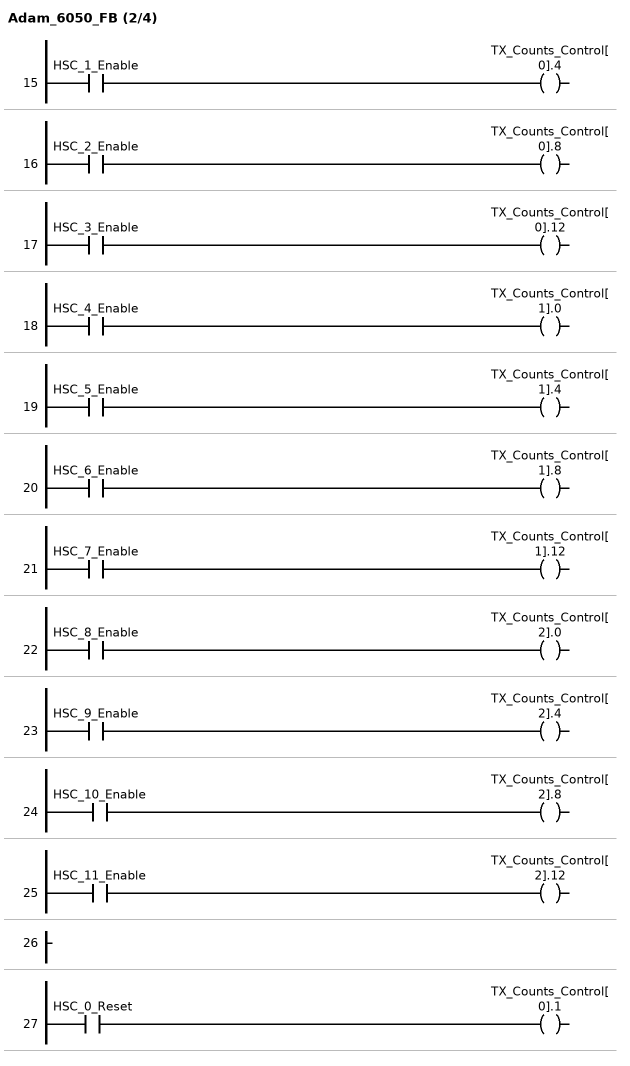
// NETWORK 15
TX_Counts_Control[0].4 := HSC_1_Enable;

// NETWORK 16
TX_Counts_Control[0].8 := HSC_2_Enable;

// NETWORK 17
TX_Counts_Control[0].12 := HSC_3_Enable;

// NETWORK 18
TX_Counts_Control[1].0 := HSC_4_Enable;

// NETWORK 19
TX_Counts_Control[1].4 := HSC_5_Enable;

// NETWORK 20
TX_Counts_Control[1].8 := HSC_6_Enable;

// NETWORK 21
TX_Counts_Control[1].12 := HSC_7_Enable;

// NETWORK 22
TX_Counts_Control[2].0 := HSC_8_Enable;

// NETWORK 23
TX_Counts_Control[2].4 := HSC_9_Enable;

// NETWORK 24
TX_Counts_Control[2].8 := HSC_10_Enable;

// NETWORK 25
TX_Counts_Control[2].12 := HSC_11_Enable;

// NETWORK 26

// NETWORK 27
TX_Counts_Control[0].1 := HSC_0_Reset;

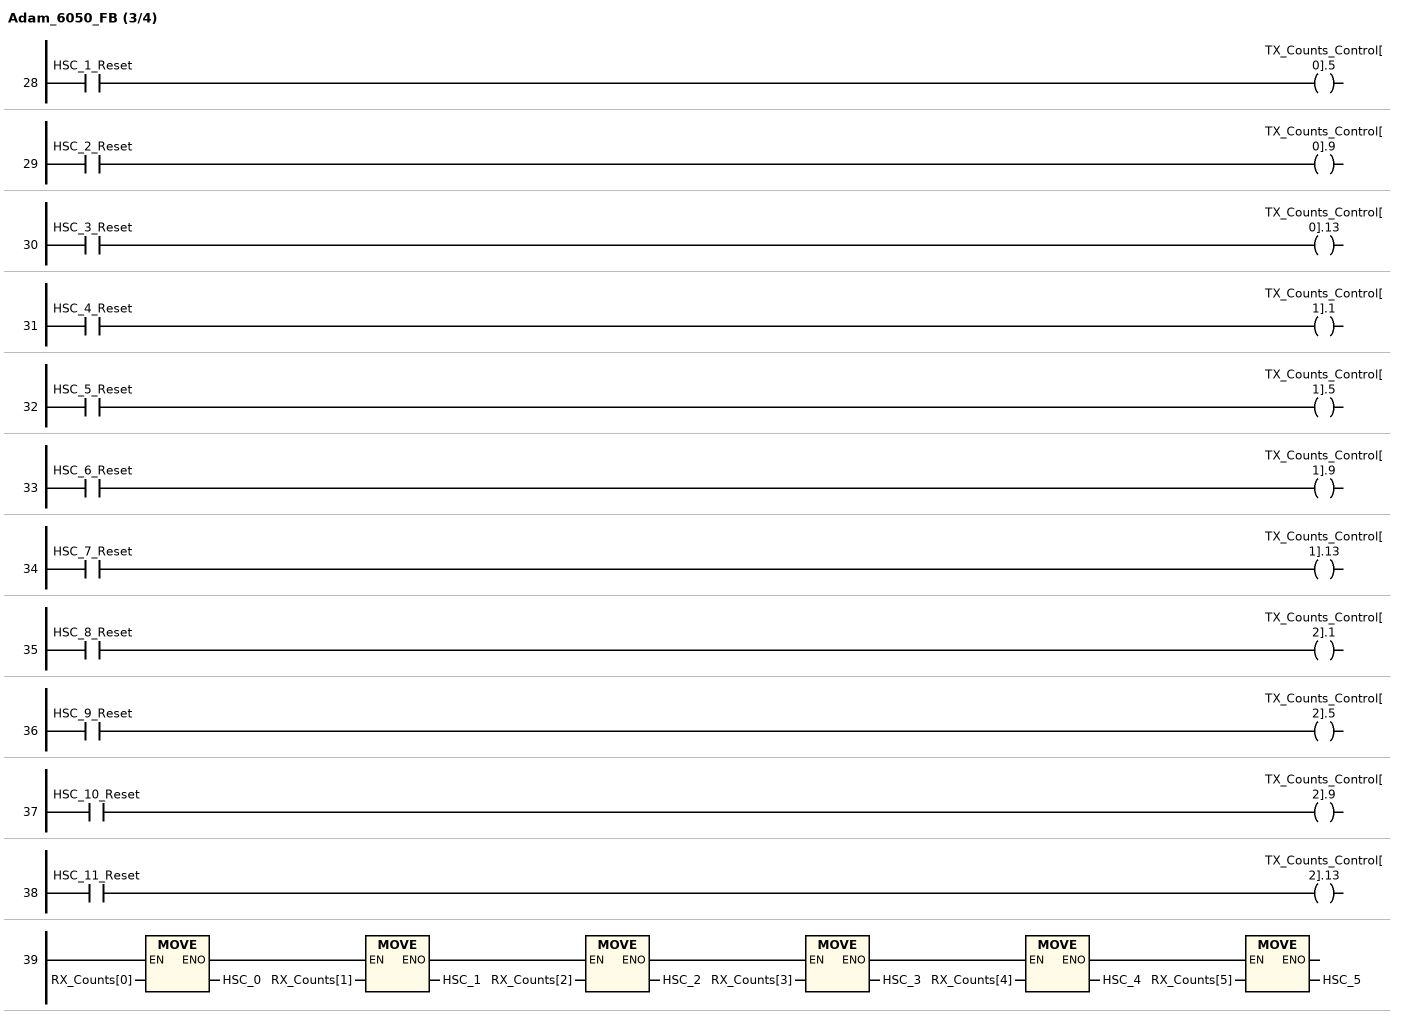
// NETWORK 28
TX_Counts_Control[0].5 := HSC_1_Reset;

// NETWORK 29
TX_Counts_Control[0].9 := HSC_2_Reset;

// NETWORK 30
TX_Counts_Control[0].13 := HSC_3_Reset;

// NETWORK 31
TX_Counts_Control[1].1 := HSC_4_Reset;

// NETWORK 32
TX_Counts_Control[1].5 := HSC_5_Reset;

// NETWORK 33
TX_Counts_Control[1].9 := HSC_6_Reset;

// NETWORK 34
TX_Counts_Control[1].13 := HSC_7_Reset;

// NETWORK 35
TX_Counts_Control[2].1 := HSC_8_Reset;

// NETWORK 36
TX_Counts_Control[2].5 := HSC_9_Reset;

// NETWORK 37
TX_Counts_Control[2].9 := HSC_10_Reset;

// NETWORK 38
TX_Counts_Control[2].13 := HSC_11_Reset;

// NETWORK 39
HSC_0 := RX_Counts[0];
HSC_1 := RX_Counts[1];
HSC_2 := RX_Counts[2];
HSC_3 := RX_Counts[3];
HSC_4 := RX_Counts[4];
HSC_5 := RX_Counts[5];

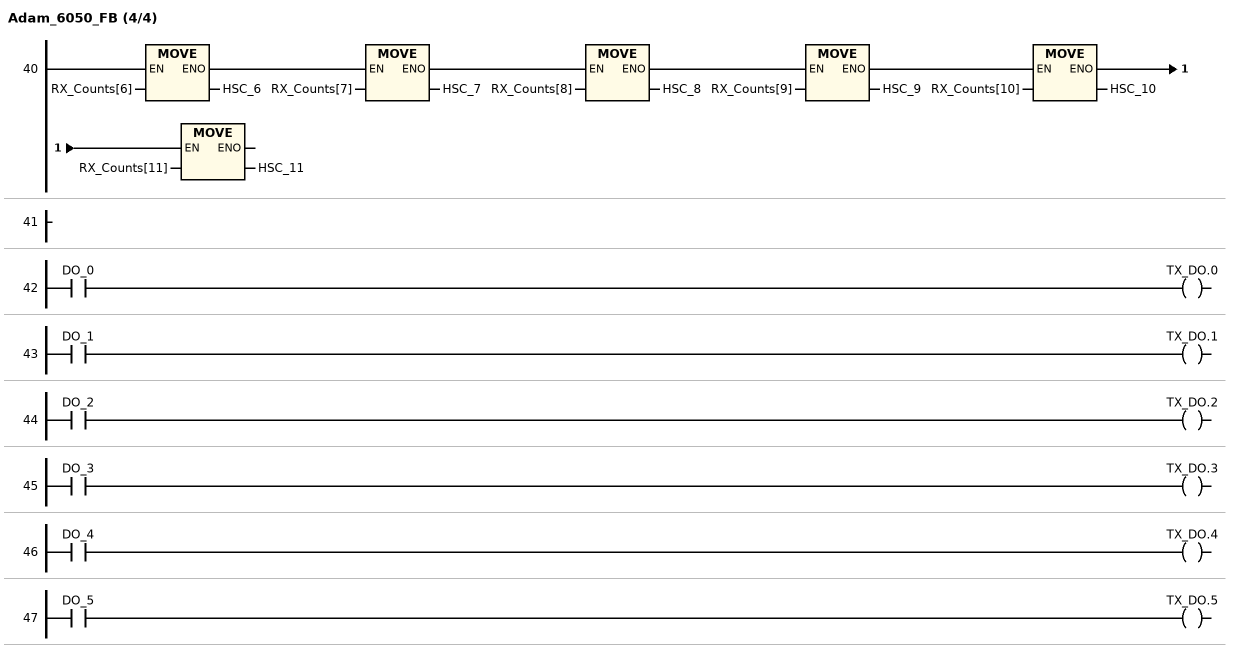
// NETWORK 40
HSC_6 := RX_Counts[6];
HSC_7 := RX_Counts[7];
HSC_8 := RX_Counts[8];
HSC_9 := RX_Counts[9];
HSC_10 := RX_Counts[10];
HSC_11 := RX_Counts[11];

// NETWORK 41

// NETWORK 42
TX_DO.0 := DO_0;

// NETWORK 43
TX_DO.1 := DO_1;

// NETWORK 44
TX_DO.2 := DO_2;

// NETWORK 45
TX_DO.3 := DO_3;

// NETWORK 46
TX_DO.4 := DO_4;

// NETWORK 47
TX_DO.5 := DO_5;

END_FUNCTION

// 20 Program Organization Units/Level_0_Remote_IO/Advantech/Adam_6217_FB
FUNCTION Adam_6217_FB : BOOL
VAR_INPUT
	RX: ARRAY[0..7] OF REAL;
	BurnOut: WORD;
	Comms_OK:BOOL;
END_VAR
VAR_OUTPUT
	AI_0:REAL;
	//AI_0_Fault:BOOL;
	AI_1:REAL;
	//AI_1_Fault:BOOL;
	AI_2:REAL;
	//AI_2_Fault:BOOL;
	AI_3:REAL;
	//AI_3_Fault:BOOL;
	AI_4:REAL;
	//AI_4_Fault:BOOL;
	AI_5:REAL;
	//AI_5_Fault:BOOL;
	AI_6:REAL;
	//AI_6_Fault:BOOL;
	AI_7:REAL;
	//AI_7_Fault:BOOL;
END_VAR
VAR
END_VAR

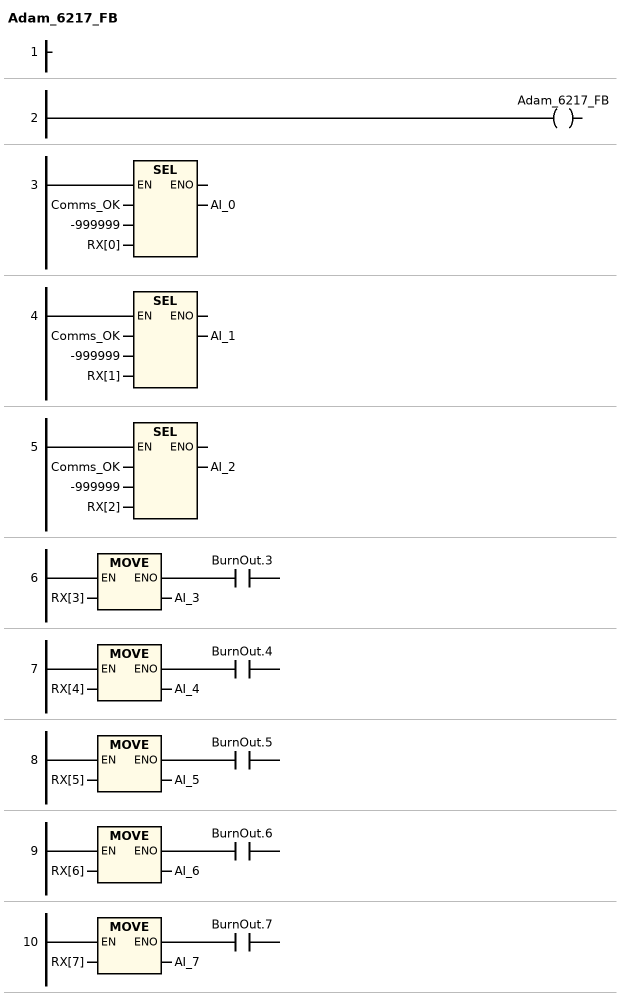
// NETWORK 1

// NETWORK 2
Adam_6217_FB := TRUE;

// NETWORK 3
AI_0 := SEL(Comms_OK, -999999, RX[0]);

// NETWORK 4
AI_1 := SEL(Comms_OK, -999999, RX[1]);

// NETWORK 5
AI_2 := SEL(Comms_OK, -999999, RX[2]);

// NETWORK 6
AI_3 := RX[3];
(* BurnOut.3; result not used *)

// NETWORK 7
AI_4 := RX[4];
(* BurnOut.4; result not used *)

// NETWORK 8
AI_5 := RX[5];
(* BurnOut.5; result not used *)

// NETWORK 9
AI_6 := RX[6];
(* BurnOut.6; result not used *)

// NETWORK 10
AI_7 := RX[7];
(* BurnOut.7; result not used *)

END_FUNCTION

// 20 Program Organization Units/Level_0_Remote_IO/Advantech/Adam_6250
FUNCTION Adam_6250 : bool
VAR_INPUT
	Device:Reference to cAdam_6250;
END_VAR
VAR
END_VAR

Device.DI[0].DI:=Device.Rx_DI.0;
Device.DI[1].DI:=Device.Rx_DI.1;
Device.DI[2].DI:=Device.Rx_DI.2;
Device.DI[3].DI:=Device.Rx_DI.3;
Device.DI[4].DI:=Device.Rx_DI.4;
Device.DI[5].DI:=Device.Rx_DI.5;
Device.DI[6].DI:=Device.Rx_DI.6;
Device.DI[7].DI:=Device.Rx_DI.7;

Device.DI[0].Count:=Device.RX_Counter_Values[0];
Device.DI[1].Count:=Device.RX_Counter_Values[1];
Device.DI[2].Count:=Device.RX_Counter_Values[2];
Device.DI[3].Count:=Device.RX_Counter_Values[3];
Device.DI[4].Count:=Device.RX_Counter_Values[4];
Device.DI[5].Count:=Device.RX_Counter_Values[5];
Device.DI[6].Count:=Device.RX_Counter_Values[6];
Device.DI[7].Count:=Device.RX_Counter_Values[7];

Device.DI[0].Frequency:=TO_REAL(Device.RX_Counter_Values[0])/10;
Device.DI[1].Frequency:=TO_REAL(Device.RX_Counter_Values[1])/10;
Device.DI[2].Frequency:=TO_REAL(Device.RX_Counter_Values[2])/10;
Device.DI[3].Frequency:=TO_REAL(Device.RX_Counter_Values[3])/10;
Device.DI[4].Frequency:=TO_REAL(Device.RX_Counter_Values[4])/10;
Device.DI[5].Frequency:=TO_REAL(Device.RX_Counter_Values[5])/10;
Device.DI[6].Frequency:=TO_REAL(Device.RX_Counter_Values[6])/10;
Device.DI[7].Frequency:=TO_REAL(Device.RX_Counter_Values[7])/10;

Device.Tx_Counter_Control[0].0:=Device.DI[0].Enable_HSC;
Device.Tx_Counter_Control[0].1:=Device.DI[1].Enable_HSC;
Device.Tx_Counter_Control[0].2:=Device.DI[2].Enable_HSC;
Device.Tx_Counter_Control[0].3:=Device.DI[3].Enable_HSC;
Device.Tx_Counter_Control[0].4:=Device.DI[4].Enable_HSC;
Device.Tx_Counter_Control[0].5:=Device.DI[5].Enable_HSC;
Device.Tx_Counter_Control[0].6:=Device.DI[6].Enable_HSC;
Device.Tx_Counter_Control[0].7:=Device.DI[7].Enable_HSC;

Device.Tx_Counter_Control[1].0:=Device.DI[0].Clear_HSC;
Device.Tx_Counter_Control[1].1:=Device.DI[1].Clear_HSC;
Device.Tx_Counter_Control[1].2:=Device.DI[2].Clear_HSC;
Device.Tx_Counter_Control[1].3:=Device.DI[3].Clear_HSC;
Device.Tx_Counter_Control[1].4:=Device.DI[4].Clear_HSC;
Device.Tx_Counter_Control[1].5:=Device.DI[5].Clear_HSC;
Device.Tx_Counter_Control[1].6:=Device.DI[6].Clear_HSC;
Device.Tx_Counter_Control[1].7:=Device.DI[7].Clear_HSC;

Device.Tx_Counter_Control[2].0:=Device.DI[0].Clear_Overflow;
Device.Tx_Counter_Control[2].1:=Device.DI[1].Clear_Overflow;
Device.Tx_Counter_Control[2].2:=Device.DI[2].Clear_Overflow;
Device.Tx_Counter_Control[2].3:=Device.DI[3].Clear_Overflow;
Device.Tx_Counter_Control[2].4:=Device.DI[4].Clear_Overflow;
Device.Tx_Counter_Control[2].5:=Device.DI[5].Clear_Overflow;
Device.Tx_Counter_Control[2].6:=Device.DI[6].Clear_Overflow;
Device.Tx_Counter_Control[2].7:=Device.DI[7].Clear_Overflow;

Device.Tx_DO.0	:=device.Dout[0].Dout;
Device.Tx_DO.1	:=device.Dout[1].Dout;
Device.Tx_DO.2	:=device.Dout[2].Dout;
Device.Tx_DO.3	:=device.Dout[3].Dout;
Device.Tx_DO.4	:=device.Dout[4].Dout;
Device.Tx_DO.5	:=device.Dout[5].Dout;
Device.Tx_DO.6	:=device.Dout[6].Dout;

Device.Tx_Pulse_Width_Low[0] :=Device.Dout[0].Pulse_Output_Low_Width;
Device.Tx_Pulse_Width_Low[1] :=Device.Dout[1].Pulse_Output_Low_Width;
Device.Tx_Pulse_Width_Low[2] :=Device.Dout[2].Pulse_Output_Low_Width;
Device.Tx_Pulse_Width_Low[3] :=Device.Dout[3].Pulse_Output_Low_Width;
Device.Tx_Pulse_Width_Low[4] :=Device.Dout[4].Pulse_Output_Low_Width;
Device.Tx_Pulse_Width_Low[5] :=Device.Dout[5].Pulse_Output_Low_Width;
Device.Tx_Pulse_Width_Low[6] :=Device.Dout[6].Pulse_Output_Low_Width;

Device.Tx_Pulse_Width_High[0]	:=Device.Dout[0].Pulse_Output_High_Width;
Device.Tx_Pulse_Width_High[1]	:=Device.Dout[1].Pulse_Output_High_Width;
Device.Tx_Pulse_Width_High[2]	:=Device.Dout[2].Pulse_Output_High_Width;
Device.Tx_Pulse_Width_High[3]	:=Device.Dout[3].Pulse_Output_High_Width;
Device.Tx_Pulse_Width_High[4]	:=Device.Dout[4].Pulse_Output_High_Width;
Device.Tx_Pulse_Width_High[5]	:=Device.Dout[5].Pulse_Output_High_Width;
Device.Tx_Pulse_Width_High[6]	:=Device.Dout[6].Pulse_Output_High_Width;

Device.Tx_Set_Absolute_Pulse[0]	:=Device.Dout[0].Set_Absolute_Pulse;
Device.Tx_Set_Absolute_Pulse[1]	:=Device.Dout[1].Set_Absolute_Pulse;
Device.Tx_Set_Absolute_Pulse[2]	:=Device.Dout[2].Set_Absolute_Pulse;
Device.Tx_Set_Absolute_Pulse[3]	:=Device.Dout[3].Set_Absolute_Pulse;
Device.Tx_Set_Absolute_Pulse[4]	:=Device.Dout[4].Set_Absolute_Pulse;
Device.Tx_Set_Absolute_Pulse[5]	:=Device.Dout[5].Set_Absolute_Pulse;
Device.Tx_Set_Absolute_Pulse[6]	:=Device.Dout[6].Set_Absolute_Pulse;

Device.Tx_Set_Incremental_Pulse[0]	:=Device.Dout[0].Set_Incremental_Pulse;
Device.Tx_Set_Incremental_Pulse[1]	:=Device.Dout[1].Set_Incremental_Pulse;
Device.Tx_Set_Incremental_Pulse[2]	:=Device.Dout[2].Set_Incremental_Pulse;
Device.Tx_Set_Incremental_Pulse[3]	:=Device.Dout[3].Set_Incremental_Pulse;
Device.Tx_Set_Incremental_Pulse[4]	:=Device.Dout[4].Set_Incremental_Pulse;
Device.Tx_Set_Incremental_Pulse[5]	:=Device.Dout[5].Set_Incremental_Pulse;
Device.Tx_Set_Incremental_Pulse[6]	:=Device.Dout[6].Set_Incremental_Pulse;

END_FUNCTION

// 20 Program Organization Units/Level_0_Remote_IO/Advantech/Adam_6266_FB
FUNCTION Adam_6266_FB : BOOL
VAR_INPUT
	HSC_0_Enable:BOOL:=FALSE;
	HSC_0_Reset:BOOL:=FALSE;
	HSC_1_Enable:BOOL:=FALSE;
	HSC_1_Reset:BOOL:=FALSE;
	HSC_2_Enable:BOOL:=FALSE;
	HSC_2_Reset:BOOL:=FALSE;
	HSC_3_Enable:BOOL:=FALSE;
	HSC_3_Reset:BOOL:=FALSE;

	
	DO_0:BOOL:=FALSE;
	DO_1:BOOL:=FALSE;
	DO_2:BOOL:=FALSE;
	DO_3:BOOL:=FALSE;

//	DO_6:BOOL;
//	DO_7:BOOL;
	RX_DI: DWORD;
	RX_Counts: ARRAY[0..3] OF UDINT;
END_VAR
VAR_OUTPUT
	HSC_0:UDINT;
	HSC_1:UDINT;
	HSC_2:UDINT;
	HSC_3:UDINT;

	
	DI_0:BOOL;
	DI_1:BOOL;
	DI_2:BOOL;
	DI_3:BOOL;

	TX_DO: WORD;
	TX_Counts_Control: WORD;
END_VAR
VAR
END_VAR

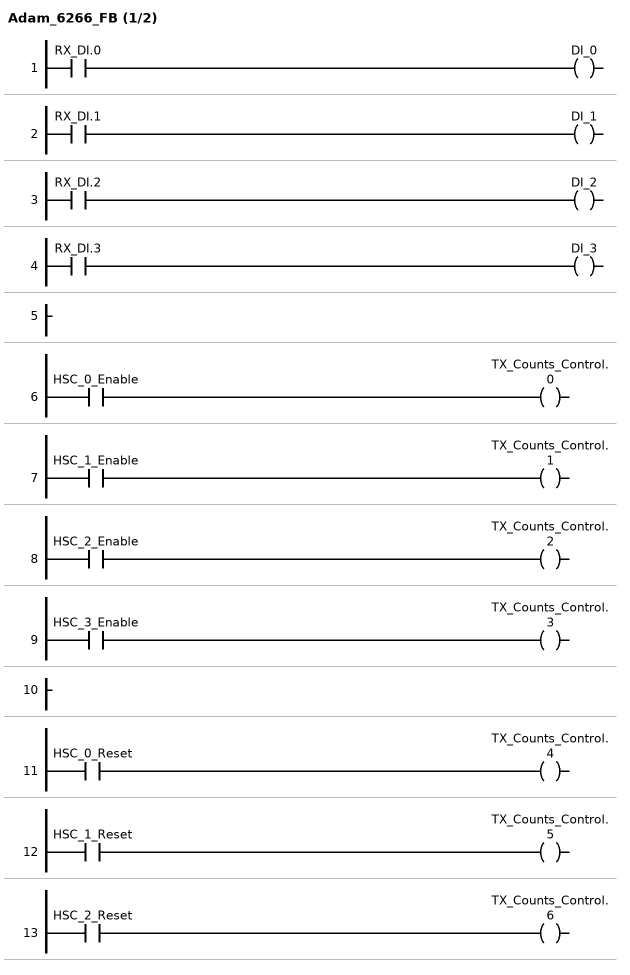
// NETWORK 1
DI_0 := RX_DI.0;

// NETWORK 2
DI_1 := RX_DI.1;

// NETWORK 3
DI_2 := RX_DI.2;

// NETWORK 4
DI_3 := RX_DI.3;

// NETWORK 5

// NETWORK 6
TX_Counts_Control.0 := HSC_0_Enable;

// NETWORK 7
TX_Counts_Control.1 := HSC_1_Enable;

// NETWORK 8
TX_Counts_Control.2 := HSC_2_Enable;

// NETWORK 9
TX_Counts_Control.3 := HSC_3_Enable;

// NETWORK 10

// NETWORK 11
TX_Counts_Control.4 := HSC_0_Reset;

// NETWORK 12
TX_Counts_Control.5 := HSC_1_Reset;

// NETWORK 13
TX_Counts_Control.6 := HSC_2_Reset;

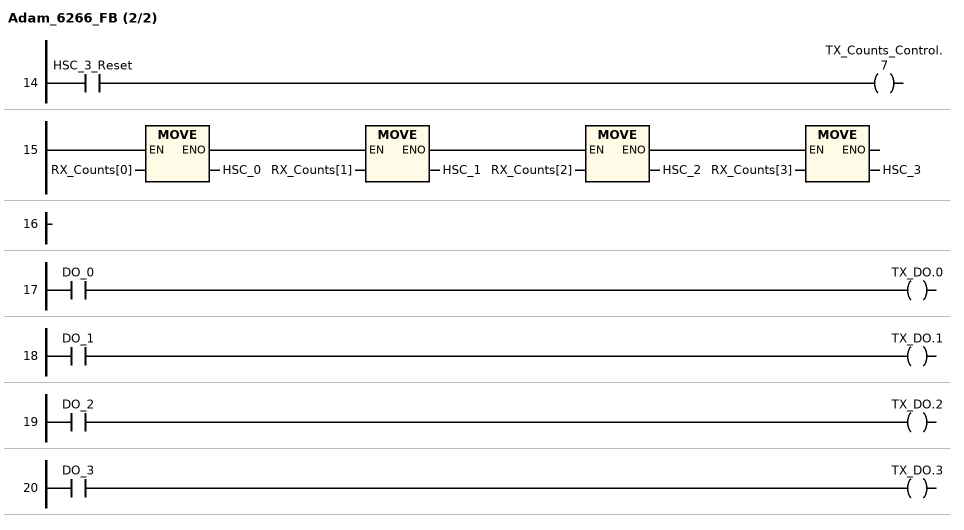
// NETWORK 14
TX_Counts_Control.7 := HSC_3_Reset;

// NETWORK 15
HSC_0 := RX_Counts[0];
HSC_1 := RX_Counts[1];
HSC_2 := RX_Counts[2];
HSC_3 := RX_Counts[3];

// NETWORK 16

// NETWORK 17
TX_DO.0 := DO_0;

// NETWORK 18
TX_DO.1 := DO_1;

// NETWORK 19
TX_DO.2 := DO_2;

// NETWORK 20
TX_DO.3 := DO_3;

END_FUNCTION

// 20 Program Organization Units/Level_0_Remote_IO/ASI/AC2916_AIT
FUNCTION_BLOCK AC2916_AIT
VAR_INPUT
	//Raw:	REAL;
	LAS:BOOL:=TRUE;
	LDS:BOOL:=TRUE;
	LPS:BOOL:=TRUE;
	LPF:BOOL:=FALSE;
	//Alarm_Enable:BOOL:=TRUE;
	//Latching:BOOL:=FALSE;
	//Fault:BOOL:=FALSE;
	Online:BOOL:=TRUE;
	Raw:WORD;
END_VAR

VAR_OUTPUT
	//Status	:BYTE;
END_VAR
VAR_IN_OUT
AIT	:	cAIT;
END_VAR

VAR(*
	hihi: BOOL;
	hi: BOOL;
	lolo: BOOL;
	LO: BOOL;
	Alarm_Debounce: TON;
	deboune_Time: TIME;
	Alarm_Active: BOOL;
	Alarm_Debounce_ET: TIME;
	Alarm: BOOL;
	ALARM_2_0: BURKERT_OSCAT_BASIC.ALARM_2;
	F_TRIG_0: F_Trig;
	TON_0: TON;
	tmpEU: REAL;
	//tmpEU1: REAL;
	tmpEU2: REAL;*)
		Analog:Analog_Sensor_UDFB;
	
END_VAR

VAR_TEMP
	//EU_Range: REAL;
	//Raw_Range: REAL;
	//Corrected_Raw: REAL;
	//Raw_Pct: REAL;
	//EU_Scaled: REAL;
END_VAR

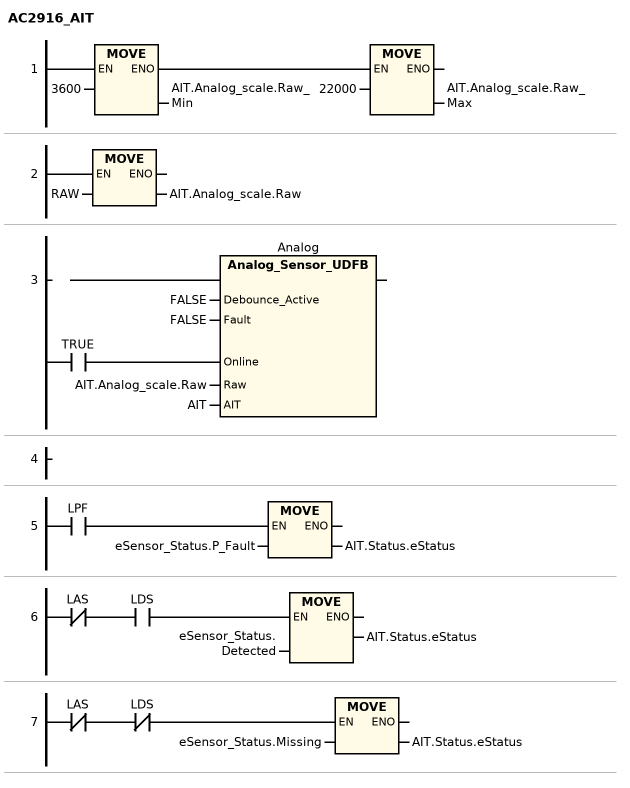
// NETWORK 1
AIT.Analog_scale.Raw_Min := 3600;
AIT.Analog_scale.Raw_Max := 22000;

// NETWORK 2
AIT.Analog_scale.Raw := RAW;

// NETWORK 3
Analog(Debounce_Active := FALSE, Fault := FALSE, Online := TRUE, Raw := AIT.Analog_scale.Raw, AIT := AIT); // Analog_Sensor_UDFB

// NETWORK 4

// NETWORK 5
IF LPF THEN AIT.Status.eStatus := eSensor_Status.P_Fault; END_IF

// NETWORK 6
IF NOT LAS AND LDS THEN AIT.Status.eStatus := eSensor_Status.Detected; END_IF

// NETWORK 7
IF NOT LAS AND NOT LDS THEN AIT.Status.eStatus := eSensor_Status.Missing; END_IF

END_FUNCTION_BLOCK

// 20 Program Organization Units/Level_1_Devices/Base_Functions/Analog_Sensor_UDFB
FUNCTION_BLOCK Analog_Sensor_UDFB
VAR_INPUT
	//Alarm_Enable:BOOL:=TRUE;
	//Latching:BOOL:=FALSE;
	Debounce_Active:Bool;
	Fault:BOOL:=FALSE;
	Online:BOOL:=TRUE;
	Raw:REAl;
END_VAR

VAR_OUTPUT
	//Status	:BYTE;
END_VAR

VAR_IN_OUT
		AIT	:	cAIT;
END_VAR

VAR
	Alarm:Analog_Alarm_UDFB;
	F_TRIG_0: F_Trig;
	TON_0: TON;
	tmpEU: REAL;
	tmpEU2: REAL;
	Valve: INT;
	Mode: INT;
	eMode: INT;
END_VAR

VAR_TEMP
	EU_Range: REAL;
	Raw_Range: REAL;
	Corrected_Raw: REAL;
	Raw_Pct: REAL;
	EU_Scaled: REAL;
END_VAR

(* body of a kind this reader does not render *)

END_FUNCTION_BLOCK

// 20 Program Organization Units/Level_0_Remote_IO/Burkert/eDip_8653_UDFB
FUNCTION eDip_8653_UDFB :BOOL
VAR_INPUT
	Node:BYTE;
	//Query:BOOL;
	
	V1:REFERENCE TO SV_DUT;
	V2:REFERENCE TO SV_DUT;
	V3:REFERENCE TO SV_DUT;
	V4:REFERENCE TO SV_DUT;
	V5:REFERENCE TO SV_DUT;
	V6:REFERENCE TO SV_DUT;
	V7:REFERENCE TO SV_DUT;
	V8:REFERENCE TO SV_DUT;
	
END_VAR
VAR_OUTPUT
END_VAR
VAR

	Data:Bytes_Dword;

END_VAR
VAR_IN_OUT
	Manifold:c8653;

	
END_VAR

(* body of a kind this reader does not render *)

END_FUNCTION

// 20 Program Organization Units/Level_0_Remote_IO/Burkert/eDip_ME64_CTRL
FUNCTION_BLOCK eDip_ME64_CTRL
VAR_INPUT
	ME64: REFERENCE TO ceDip_ME64_DUT;
	Node:Byte;
END_VAR
VAR_OUTPUT
END_VAR
VAR
	Data:Bytes_Dword;
END_VAR

ME64.DSO.Node:=Node;
Parse_RX();
Parse_TX();

END_FUNCTION_BLOCK

// 20 Program Organization Units/Level_0_Remote_IO/Burkert/eDip_ReadDDO
FUNCTION_BLOCK eDip_ReadDDO
VAR_INPUT
	ReadSingleItem : REFERENCE TO eDip_ReadSingleItem;
	DDO: REFERENCE TO cDDO;
	Enable:BOOL;
	
END_VAR
VAR_OUTPUT
	Complete:BOOL;
END_VAR
VAR
	Stage:BYTE:=0;
END_VAR

IF NOT(Enable) THEN
	Complete:=FALSE;
	Stage:=0;
END_IF

CASE Stage OF
	0:	IF Enable THEN Stage:=1;END_IF;
	1:	ReadSingleItem.Index:=16#1018;
		ReadSingleItem.SubIndex:=16#02;
		ReadSingleItem.Enable:=TRUE;
		Stage:=Stage+1;
	2:	IF ReadSingleItem.Complete THEN
			DDO.Product_Code:=ReadSingleItem.Data.tDword;
			ReadSingleItem.Enable:=FALSE;
			Stage:=Stage+1;
		END_IF;
	3:	ReadSingleItem.Index:=16#1018;
		ReadSingleItem.SubIndex:=16#04;
		ReadSingleItem.Enable:=TRUE;
		Stage:=Stage+1;
	4:	IF ReadSingleItem.Complete THEN
			DDO.Serial_Number:=ReadSingleItem.Data.tDword;
			ReadSingleItem.Enable:=FALSE;
			Stage:=Stage+1;
		END_IF
	5:	ReadSingleItem.Index:=16#2000;
		ReadSingleItem.SubIndex:=16#02;
		ReadSingleItem.Enable:=TRUE;
		Stage:=Stage+1;
	6:	IF ReadSingleItem.Complete THEN
			DDO.Ident:=ReadSingleItem.Data.tDword;
			ReadSingleItem.Enable:=FALSE;
			Stage:=Stage+1;
		END_IF
		
	7:	ReadSingleItem.Enable:=FALSE;
		Complete:=TRUE;
END_CASE;

END_FUNCTION_BLOCK

// 20 Program Organization Units/Level_0_Remote_IO/Burkert/eDip_ReadSingleItem
FUNCTION_BLOCK eDip_ReadSingleItem
VAR_INPUT
    Index     : WORD;
    SubIndex  : BYTE;
    Node      : BYTE;
	Enable:BOOL;
	orf:REFERENCE TO eDip_MEx3_ORF;
END_VAR
VAR_OUTPUT
	Data:Bytes_Dword;
	Complete:BOOL;
END_VAR
VAR
	Stage:BYTE:=0;
	Flash:Burkert_OSCAT_BASIC.GEN_PULSE;
	Active_count:UINT:=0;
	Fault_Count:UINT:=0;
	Fault_Code:DWORD;
	Raw_Data:Dword;
	
END_VAR

Flash(ENQ:=TRUE,PTH:=T#50MS,PTL:=T#50MS);

IF NOT(Enable) THEN Stage:=0; END_IF

CASE Stage OF
	0:	Complete:=FALSE;
		Raw_Data:=16#FFFFFFFE;
		IF Enable THEN 
			Stage:=1;
			//ORF.Write_Value:=FALSE;
			END_IF
	1:	//Clear Old Data
		ORF.Call := 0;
        ORF.Length := 16#00040000;
        ORF.Value_TX := 16#FFFFFFFF;
		ORF.Index_TX:=Build_Orf_Index(Index:=Index,SubIndex:=SubIndex,Node:=Node,Write:=FALSE);
		ORF.Write_Value:=FALSE;
		Stage:=2;
	2:	ORF.Write_Value:=TRUE;
		Stage:=3;

	3:	ORF.Write_Value:=Flash.Q;
		IF ORF.Index_RX=ORF.Index_TX AND ORF.Value_RX=16#FFFFFFFF	 THEN 
			ORF.Length := 16#0000;
			ORF.Write_Value:=FALSE;
			Orf.Call.8:=TRUE;
			Stage:=6;
		END_IF;
(*
	4: 	Orf.Call.8:=Flash.Q;
		IF Flash.Q THEN Stage:=5; END_IF;
	5: 	IF NOT(Flash.Q) THEN Stage:=6; END_IF;
*)
	6:	Raw_Data:=ORF.Value_RX;
		IF Raw_Data<16#FFFFFFFE	THEN 
			Data.tDword:=MEM.ReverseWORDsInDWORD(dwInput:=Raw_Data );
			Stage:=7; 
		END_IF;
		Orf.Call.8:=TRUE;
		IF ORF.Result=16#FFFFFFFF THEN Active_count:=Active_count+1; END_IF;
		IF ORF.Result>1 AND ORF.Result<16#FFFFFFFF AND Flash.Q	THEN Stage:=9; END_IF;
		
	7:	//First_data:=MEM.ReverseWORDsInDWORD(dwInput:=orf.Value_RX );
		ORF.Value_TX:=0;
		Orf.Call:=16#0000;
		ORF.Write_Value:=FALSE;
		Raw_Data:=16#FFFFFFFD;
		Stage:=8;
	8:	
		Complete:=TRUE;
		ORF.Write_Value:=FALSE;
		Orf.Call:=16#0000;		
	9: 
		Fault_Code:=MEM.ReverseWORDsInDWORD(dwInput:=orf.Result );
		Data.tDword:=0;
		ORF.Index_TX:=Build_Orf_Index(Index:=16#1000,SubIndex:=16#0,Node:=Node,Write:=FALSE);
		Fault_Count:=Fault_Count+1;
		Stage:=10;
	10:
		Orf.Call.8:=Flash.Q;
		IF orf.Result=0 THEN stage:=11;END_IF;
	11:	Orf.Call:=0;
		ORF.Index_TX:=Build_Orf_Index(Index:=Index,SubIndex:=SubIndex,Node:=Node,Write:=FALSE);
		Complete:=TRUE;
END_CASE

END_FUNCTION_BLOCK

// 20 Program Organization Units/Level_0_Remote_IO/Burkert/eDip_ReadDSO
FUNCTION_BLOCK eDip_ReadDSO
VAR_INPUT
	ReadSingleItem : REFERENCE TO eDip_ReadSingleItem;
	DSO: REFERENCE TO cDSO;
	Enable:BOOL;
	
END_VAR
VAR_OUTPUT
	Complete:BOOL;
END_VAR
VAR
	Stage:BYTE:=0;
END_VAR

IF NOT(Enable) THEN
	Complete:=FALSE;
	Stage:=0;
END_IF

CASE Stage OF
	0:	IF Enable THEN Stage:=1;END_IF;
	1:	ReadSingleItem.Index:=16#2004;
		ReadSingleItem.SubIndex:=16#01;
		ReadSingleItem.Enable:=TRUE;
		Stage:=Stage+1;
	2:	IF ReadSingleItem.Complete THEN
			DSO.NamurNe107.iNamur:=ReadSingleItem.Data.tByte[0];
			ReadSingleItem.Enable:=FALSE;
			Stage:=Stage+1;
		END_IF;
	3:	ReadSingleItem.Index:=16#2004;
		ReadSingleItem.SubIndex:=16#02;
		ReadSingleItem.Enable:=TRUE;
		Stage:=Stage+1;
	4:	IF ReadSingleItem.Complete THEN
			DSO.Temperature:=ReadSingleItem.Data.tReal;
			ReadSingleItem.Enable:=FALSE;
			Stage:=Stage+1;
		END_IF
	5:	ReadSingleItem.Index:=16#2004;
		ReadSingleItem.SubIndex:=16#03;
		ReadSingleItem.Enable:=TRUE;
		Stage:=Stage+1;
	6:	IF ReadSingleItem.Complete THEN
			DSO.Voltage:=ReadSingleItem.Data.tReal;
			ReadSingleItem.Enable:=FALSE;
			Stage:=Stage+1;
		END_IF
	7:	ReadSingleItem.Index:=16#2004;
		ReadSingleItem.SubIndex:=16#04;
		ReadSingleItem.Enable:=TRUE;
		Stage:=Stage+1;
	8:	IF ReadSingleItem.Complete THEN
			DSO.Operation_Time:=ReadSingleItem.Data.tUDINT;
			ReadSingleItem.Enable:=FALSE;
			Stage:=Stage+1;
		END_IF
		
		
		
	9:	ReadSingleItem.Enable:=FALSE;
		Complete:=TRUE;
END_CASE;

END_FUNCTION_BLOCK

// 20 Program Organization Units/Level_0_Remote_IO/Burkert/eDip_WriteSingleItem
FUNCTION_BLOCK eDip_WriteSingleItem
VAR_INPUT
    Index     : WORD;
    SubIndex  : BYTE;
    Node	: BYTE;
	Length	: BYTE;
	Data	:Bytes_Dword;
	Enable:BOOL;
	orf:REFERENCE TO eDip_MEx3_ORF;
END_VAR
VAR_OUTPUT
	Complete:BOOL;
END_VAR
VAR
	Stage:BYTE:=0;
	Flash:Burkert_OSCAT_BASIC.GEN_PULSE;
	TX_Dword:Dword;
	
END_VAR

Flash(ENQ:=TRUE,PTH:=T#100MS,PTL:=T#100MS);

IF NOT(Enable) THEN Stage:=0; END_IF
tx_Dword:=MEM.ReverseWORDsInDWORD(dwInput:=Data.tDword );
CASE Stage OF
	0:	Complete:=FALSE;
		IF Enable THEN 
			Stage:=1;
			//ORF.Write_Value:=FALSE;
			END_IF
	1:	
		ORF.Call := 0;
        ORF.Length := Length *16#10000;
        ORF.Value_TX := tx_Dword;
		ORF.Index_TX:=Build_Orf_Index(Index:=Index,SubIndex:=SubIndex,Node:=Node,Write:=TRUE);
		ORF.Write_Value:=FALSE;
		Stage:=2;
	2:	ORF.Write_Value:=TRUE;
		Stage:=3;

	3:	ORF.Write_Value:=Flash.Q;
		IF ORF.Index_RX=ORF.Index_TX AND ORF.Value_RX=tx_Dword	 THEN 
			ORF.Write_Value:=FALSE;
			IF Flash.Q THEN	Orf.Call.8:=TRUE; END_IF;
			IF ORF.Call.8 AND NOT(Flash.Q) THEN	Stage:=4; END_IF;
		END_IF;

	4:	IF ORF.Result=0 AND Flash.Q	THEN Stage:=5; END_IF;

	5:	
		Complete:=TRUE;
		ORF.Write_Value:=FALSE;
		Orf.Call:=16#0000;
		ORF.Length := 16#0000;		

END_CASE

END_FUNCTION_BLOCK

// 20 Program Organization Units/Level_0_Remote_IO/Burkert/ME43_SDO
FUNCTION_BLOCK ME43_SDO
VAR_INPUT
	CommState:	ModbusTCPComState;
	Node:	BYTE;
	orf:	REFERENCE TO eDip_MEx3_ORF;
	
	
	r8228:	REFERENCE TO ceDip_8228;
	r8312: 	REFERENCE TO c8312;
	r8412: 	REFERENCE TO c8412;
	r8691:	REFERENCE TO cDigital_BCV;
	r8694:	REFERENCE TO cDigital_ACV;
	r8653:	REFERENCE TO c8653;
	rME64:	REFERENCE TO cME64;
	r8098:	REFERENCE TO c8098;
	r336x:	REFERENCE TO c336x;
	
	rME44AI:REFERENCE TO cME44_AI;
	
	
END_VAR
VAR_OUTPUT
	Product_Code:DWORD;
	Result:DWORD;
	
END_VAR
VAR
	
Task:eMEx3SDO;
//uORF:Bytes_Dword;
Value:Bytes_Dword;
Pulse:Burkert_OSCAT_BASIC.CLK_PRG;
Active:ARRAY[0..127] OF DWORD;
Scan_Index:UINT;
Device_Stage:UINT;
Scan_Clear_Count:DWORD;

SubStage:BYTE;
Flash:Burkert_OSCAT_BASIC.GEN_PULSE;
Reset_R_trig:R_trig;

ORF_Stage:BYTE:=0;
data:Bytes_Dword;
dio:cDIO;
DSO:cDSO;
DDO:cDDO;


ReadSingleItem:eDip_ReadSingleItem;

WriteSingleItem:eDip_WriteSingleItem;
ReadDDO :eDip_ReadDDo;
ReadDSO :eDip_ReadDSO;

Direct_Write_R_trig:R_trig;
t8312:c8312;
t8412:c8412;
t8691:cDigital_BCV;
t8694:cDigital_ACV;
t8653:c8653;
t8228:ceDip_8228;
tME44AI:cME44_AI;
tME64:cME64;
t8098:c8098;
t336x:c336x;

END_VAR

//0x10180-02 Product Code
orf.CommState:=CommState;
CASE CommState OF
	ModbusTCPComState.OFF: ORF.strTCPstate:='OFF';
	ModbusTCPComState.CONNECTING: ORF.strTCPstate:='CONNECTING';
	ModbusTCPComState.CONNECTED: ORF.strTCPstate:='CONNECTED';
	ModbusTCPComState.DISCONNECTING: ORF.strTCPstate:='DISCONNECTING';
	ModbusTCPComState.SOCKET_ERROR: ORF.strTCPstate:='SOCKET_ERROR';
END_CASE

IF WriteSingleItem.Enable THEN ReadSingleItem.Enable:=FALSE; END_IF;


ReadSingleItem(Node:=Node,orf:=orf);
WriteSingleItem(orf:=orf);
//WriteSingleItem();

ReadDDO(ReadSingleItem:=ReadSingleItem);
ReadDSO(ReadSingleItem:=ReadSingleItem);

Pulse(PT:=T#500MS);
Flash(ENQ:=TRUE,PTH:=T#250MS,PTL:=T#250MS);
Result:=ORF.Value_RX;
Direct_Write_R_trig();
//ORF.Index:=uORF.tDword;

Reset_R_trig(clk:=(Node>127 OR Node=0));
IF Reset_r_trig.Q THEN	
	ReadSingleItem.Enable:=FALSE;
	WriteSingleItem.Enable:=FALSE;
	orf.Control_Word.tWord[0]:=0;
	orf.Control_Word.tWord[1]:=0;
	orf.Restart:=FALSE;
END_IF;
IF Node>127 OR Node=0  THEN 

	Task:=eMEx3SDO.Idle;
	ReadSingleItem.Enable:=FALSE;
	//WriteSingleItem.Enable:=FALSE;
	product_Code:=0;
	Device_Stage:=0;
	//orf.Call:=16#00;
	//ORF.Write_Value:=FALSE;
	ReadDDO.Enable:=FALSE;
	ReadDSO.Enable:=FALSE;
ELSE
	//Direct_Write.Node:=Node;
	//Direct_Write.orf:=Orf;
	
	IF Product_code=0 OR product_code>16#FFFFFFFA THEN
		ReadSingleItem.Index := 16#1018;
		ReadSingleItem.SubIndex := 16#02;
		ReadSingleItem.Enable:=TRUE;
		IF ReadSingleItem.Complete THEN 
			Product_Code:=ReadSingleItem.Data.tDword;
			ReadSingleItem.Enable:=FALSE;
		END_IF;
	END_IF;
END_IF;


IF ORF.Result=16#FFFFFFFF THEN Orf.Call:=0;END_IF;

CASE product_code OF
	0:		SubStage:=0;Device_Stage:=0;
	8228: 		edip_8228();
	8653: 		edip_8653();
	8691: 		edip_8691();
	8694:		eDip_8694();
	8695: 		edip_8695();
	8098:		s8098();
	3363:		eDip_336x();
	1296380980 	:ME44_AI();
	1296381492	:ME64();
	
	
	16#FFFFFFFA:	SubStage:=0;Device_Stage:=0;
		
	
	
END_CASE;


IF Node>127 OR Node=0 THEN
	IF orf.Restart=TRUE THEN
		IF orf.CommState=ModbusTCPComState.CONNECTED THEN
			orf.Control_Word.tWord[0]:=16#8100;
			orf.Control_Word.tWord[1]:=16#0100;
		ELSE
			orf.Control_Word.tWord[0]:=0;
			orf.Control_Word.tWord[1]:=0;
			orf.Restart:=FALSE;
		END_IF;
	END_IF;
END_IF;

END_FUNCTION_BLOCK

// 20 Program Organization Units/Level_0_Remote_IO/Burkert/ME44_DI
FUNCTION ME44_DI :BOOL;
VAR_INPUT
		device :REFERENCE TO cME44_DI;
		Node:BYTE;
END_VAR
VAR
	//Data:Bytes_Dword;
END_VAR

Device.DSO.Node:=Node;(*
Device.Namur:=Device.RX.Namur.tByte[1];

Device.Ch[1].Hz_Count:=Device.RX.DI1_Float.tReal;
Device.Ch[2].Hz_Count:=Device.RX.DI2_Float.tReal;
Device.Ch[3].Hz_Count:=Device.RX.DI3_Float.tReal;
Device.Ch[4].Hz_Count:=Device.RX.DI4_Float.tReal;
Device.Ch[5].Hz_Count:=Device.RX.DI5_Float.tReal;
Device.Ch[6].Hz_Count:=Device.RX.DI6_Float.tReal;
Device.Ch[7].Hz_Count:=Device.RX.DI7_Float.tReal;
Device.Ch[8].Hz_Count:=Device.RX.DI8_Float.tReal;

Device.Ch[1].Totaliser:=Device.RX.DI1_Total.tReal;
Device.Ch[2].Totaliser:=Device.RX.DI2_Total.tReal;
Device.Ch[3].Totaliser:=Device.RX.DI3_Total.tReal;
Device.Ch[4].Totaliser:=Device.RX.DI4_Total.tReal;
Device.Ch[5].Totaliser:=Device.RX.DI5_Total.tReal;
Device.Ch[6].Totaliser:=Device.RX.DI6_Total.tReal;
Device.Ch[7].Totaliser:=Device.RX.DI7_Total.tReal;
Device.Ch[8].Totaliser:=Device.RX.DI8_Total.tReal;

Device.Ch[1].Raw:=Device.RX.DI1_DI_8.tByte[1].0;
Device.Ch[2].Raw:=Device.RX.DI1_DI_8.tByte[1].1;
Device.Ch[3].Raw:=Device.RX.DI1_DI_8.tByte[1].2;
Device.Ch[4].Raw:=Device.RX.DI1_DI_8.tByte[1].3;
Device.Ch[5].Raw:=Device.RX.DI1_DI_8.tByte[1].4;
Device.Ch[6].Raw:=Device.RX.DI1_DI_8.tByte[1].5;
Device.Ch[7].Raw:=Device.RX.DI1_DI_8.tByte[1].6;
Device.Ch[8].Raw:=Device.RX.DI1_DI_8.tByte[1].7;





Device.TX.Counter_Reset.8:=Device.Ch[1].Reset_Count;
Device.TX.Totaliser_Reset.8:=Device.Ch[1].Reset_Totaliser;

Device.TX.Counter_Reset.9:=Device.Ch[2].Reset_Count;
Device.TX.Totaliser_Reset.9:=Device.Ch[2].Reset_Totaliser;

Device.TX.Counter_Reset.10:=Device.Ch[3].Reset_Count;
Device.TX.Totaliser_Reset.10:=Device.Ch[3].Reset_Totaliser;

Device.TX.Counter_Reset.11:=Device.Ch[4].Reset_Count;
Device.TX.Totaliser_Reset.11:=Device.Ch[4].Reset_Totaliser;

Device.TX.Counter_Reset.12:=Device.Ch[5].Reset_Count;
Device.TX.Totaliser_Reset.12:=Device.Ch[5].Reset_Totaliser;

Device.TX.Counter_Reset.13:=Device.Ch[6].Reset_Count;
Device.TX.Totaliser_Reset.13:=Device.Ch[6].Reset_Totaliser;

Device.TX.Counter_Reset.14:=Device.Ch[7].Reset_Count;
Device.TX.Totaliser_Reset.14:=Device.Ch[7].Reset_Totaliser;

Device.TX.Counter_Reset.15:=Device.Ch[8].Reset_Count;
Device.TX.Totaliser_Reset.15:=Device.Ch[8].Reset_Totaliser;

*)

END_FUNCTION

// 20 Program Organization Units/Level_0_Remote_IO/CanOpen/CanOpen_8605
FUNCTION_BLOCK CanOpen_8605
VAR_INPUT
	CanOpen:	REFERENCE TO _3SCOS.CANRemoteDevice_Diag;
	Device:		REFERENCE TO cCanOpen_8605;
	
END_VAR
VAR_OUTPUT
END_VAR
VAR
	SDO_CLK:Burkert_OSCAT_BASIC.CLK_PRG;
	AutoRead_CLK:Burkert_OSCAT_BASIC.CLK_PRG;
	
	SDO_Read:CIA405.SDO_READ4;
	SDO_Write:CIA405.SDO_WRITE_DATA;
	
END_VAR

CanOpen_NMT();
IF Device.CanOpen.Device_State=_3SCOS.DED.DEVICE_STATE.RUNNING THEN
	AutoRead_CLK(PT:=T#30S);
	SDO_CLK(PT:=T#200MS);
	IF Device.CanOpen.Read_Once THEN
		READ_SDO();
	ELSE
		Write_SDO();
	END_IF
END_IF

IF AutoRead_CLK.Q THEN
	Device.CanOpen.Read_Once:=TRUE;
END_IF

//Device.pdo.Namur.iNamur:=Device.PDO.Namur;
Device.DSO.StrNamur:=Burkert_OSCAT_BASIC.REPLACE_ALL(str:=TO_STRING(Device.pdo.Namur.eNamur) , src:='_' , rep:=' ' );

END_FUNCTION_BLOCK

// 20 Program Organization Units/Level_0_Remote_IO/CanOpen/CanOpen_8653
FUNCTION_BLOCK CanOpen_8653
VAR_INPUT
	V1:REFERENCE TO SV_DUT;
	V2:REFERENCE TO SV_DUT;
	V3:REFERENCE TO SV_DUT;
	V4:REFERENCE TO SV_DUT;
	V5:REFERENCE TO SV_DUT;
	V6:REFERENCE TO SV_DUT;
	V7:REFERENCE TO SV_DUT;
	V8:REFERENCE TO SV_DUT;
	
	CanOpen:	REFERENCE TO _3SCOS.CANRemoteDevice_Diag;
	Device:		REFERENCE TO cCanOpen_8653;
END_VAR
VAR_OUTPUT
END_VAR
VAR
	SDO_CLK:Burkert_OSCAT_BASIC.CLK_PRG;
	AutoRead_CLK:Burkert_OSCAT_BASIC.CLK_PRG;
	
	SDO_Read:CIA405.SDO_READ4;
	SDO_Write:CIA405.SDO_WRITE_DATA;
	
END_VAR

CanOpen_NMT();
SV_Mapping();


//Device.cPDO.Namur.iNamur:=Device.PDO.NamurStatus;
Device.DSO.StrNamur:=Burkert_OSCAT_BASIC.REPLACE_ALL(str:=TO_STRING(Device.PDO.Namur.eNamur) , src:='_' , rep:=' ' );


IF Device.CanOpen.Device_State=_3SCOS.DED.DEVICE_STATE.RUNNING THEN
	Device.Ready:=TRUE;
	AutoRead_CLK(PT:=T#60S);
	SDO_CLK(PT:=T#200MS);
	PDO_TX();
	IF Device.CanOpen.Read_Once THEN
		READ_SDO();
	ELSE
		Write_SDO();
	END_IF
ELSE
	Device.Ready:=FALSE;
	Device.PDO.Namur.iNamur:=10;//eNamur107.Offline;
END_IF

IF AutoRead_CLK.Q THEN
	Device.CanOpen.Read_Once:=TRUE;
END_IF

END_FUNCTION_BLOCK

// 20 Program Organization Units/Level_0_Remote_IO/CanOpen/CanOpen_ME64
FUNCTION_BLOCK CanOpen_ME64
VAR_INPUT
	CanOpen:	REFERENCE TO _3SCOS.CANRemoteDevice_Diag;
	Device:		REFERENCE TO cCanOpen_ME64;
	
	X1_A_FIT:REFERENCE TO cBase_FIT;
	X1_B_FIT:REFERENCE TO cBase_FIT;
	X5_A_FIT:REFERENCE TO cBase_FIT;
	X5_B_FIT:REFERENCE TO cBase_FIT;
END_VAR
VAR_OUTPUT
END_VAR
VAR
	SDO_CLK:Burkert_OSCAT_BASIC.CLK_PRG;
	AutoRead_CLK:Burkert_OSCAT_BASIC.CLK_PRG;
	
	SDO_Read:CIA405.SDO_READ4;
	SDO_Write:CIA405.SDO_WRITE_DATA;
	
END_VAR

CanOpen_NMT();
PDO_TX();
Build_PDO();

//Device.cpoNamur.iNamur:=Device.PDO.NamurStatus;
//Device.DSO.StrNamur:=Burkert_OSCAT_BASIC.REPLACE_ALL(str:=TO_STRING(Device.DSO.Namur.eNamur) , src:='_' , rep:=' ' );

IF Device.CanOpen.Device_State=_3SCOS.DED.DEVICE_STATE.RUNNING THEN
	AutoRead_CLK(PT:=T#30S);
	SDO_CLK(PT:=T#200MS);
	SDO_READ(Index:=Device.CanOpen.Index,SubIndex:=Device.CanOpen.SubIndex,Data=>Device.CanOpen.Data.tByte);
	//Parse_SDO();

	IF Device.CanOpen.Read_Once THEN
		READ_SDO();
	ELSE
		Write_SDO();
	END_IF
END_IF

IF AutoRead_CLK.Q THEN
	Device.CanOpen.Read_Once:=TRUE;
END_IF

END_FUNCTION_BLOCK

// 20 Program Organization Units/Level_0_Remote_IO/eDip/eDip_8605_CTRL
FUNCTION_BLOCK eDip_8605_CTRL
VAR_INPUT
	GW_TCP_State:ModbusTCPComState;
	Device: REFERENCE TO ceDip_8605;
	Node:BYTE;
	//Inhibit:BOOL;
	Kick_Active:BOOL;
END_VAR
VAR_OUTPUT
	Kick_Request:BOOL;
END_VAR
VAR
	//Data:Bytes_Dword;
	Last_DO_State:BOOL;
	Kick_TP:TP;
	Kick_Delay:TON;
END_VAR

Kick_delay(PT:=T#1S);
Kick_TP(PT:=T#1S,In:=Device.TX.8);

Parse_RX();
Parse_TX();
Last_Do_State:=Device.TX.8;

Device.DSO.Node:=Node;

CASE GW_TCP_State OF
	ModbusTCPComState.OFF: Device.strTCPstate:='OFF';
	ModbusTCPComState.CONNECTING: Device.strTCPstate:='CONNECTING';
	ModbusTCPComState.CONNECTED: Device.strTCPstate:='CONNECTED';
	ModbusTCPComState.DISCONNECTING: Device.strTCPstate:='DISCONNECTING';
	ModbusTCPComState.SOCKET_ERROR: Device.strTCPstate:='SOCKET_ERROR';
END_CASE

END_FUNCTION_BLOCK

// 20 Program Organization Units/Level_0_Remote_IO/eDip/eDip_ME44_AI
FUNCTION eDip_ME44_AI :BOOL
VAR_INPUT
	Device: REFERENCE TO ceDip_ME44_AI;
	Node:BYTE;
	GW_TCP_State:ModbusTCPComState;
END_VAR
VAR_OUTPUT
	Ready:Bool;
END_VAR
VAR
	Data:Bytes_Dword;
END_VAR

Device.DSO.Node:=Node;
IF GW_TCP_State=ModbusTCPComState.CONNECTED THEN
	Ready:=TRUE;
	Device.Namur.iNamur:=Device.RX.Namur.tByte[1];
	Device.AI[1]:=Device.RX.CH1.tReal;
	Device.AI[2]:=Device.RX.CH2.tReal;
	Device.AI[3]:=Device.RX.CH3.tReal;
	Device.AI[4]:=Device.RX.CH4.tReal;
ELSE
	Device.Namur.eNamur:=eNamur107.Offline;
	Ready:=FALSE;
	Device.AI[1]:=0;
	Device.AI[2]:=0;
	Device.AI[3]:=0;
	Device.AI[4]:=0;
END_IF;





CASE GW_TCP_State OF
	ModbusTCPComState.OFF: Device.strTCPstate:='OFF';
	ModbusTCPComState.CONNECTING: Device.strTCPstate:='CONNECTING';
	ModbusTCPComState.CONNECTED: Device.strTCPstate:='CONNECTED';
	ModbusTCPComState.DISCONNECTING: Device.strTCPstate:='DISCONNECTING';
	ModbusTCPComState.SOCKET_ERROR: Device.strTCPstate:='SOCKET_ERROR';
END_CASE



Device.DSO.StrNamur:=Burkert_OSCAT_BASIC.REPLACE_ALL(str:=TO_STRING(Device.DSO.NamurNe107.eNamur) , src:='_' , rep:=' ' );

END_FUNCTION

// 20 Program Organization Units/Level_0_Remote_IO/eDip/eDip_ME44_AO
FUNCTION eDip_ME44_AO : bool
VAR_INPUT
	Device: REFERENCE TO cME44_AO;
	
	CH1:REAL;
	CH2:REAL;
	CH3:REAL;
	CH4:REAL;
END_VAR
VAR
	Data:Bytes_Dword;
END_VAR

Device.AO[1]:=Ch1;
Device.AO[2]:=Ch2;
Device.AO[3]:=Ch3;
Device.AO[4]:=Ch4;


Data.tWord[0]:=Device.RX_Namur;
Device.Namur:=Data.tByte[1];

Data.tReal:=Device.AO[1];
Device.TX.CH1[0]:=Data.tWord[0];
Device.TX.CH1[1]:=Data.tWord[1];

Data.tReal:=Device.AO[2];
Device.TX.CH2[0]:=Data.tWord[0];
Device.TX.CH2[1]:=Data.tWord[1];

Data.tReal:=Device.AO[3];
Device.TX.CH3[0]:=Data.tWord[0];
Device.TX.CH3[1]:=Data.tWord[1];

Data.tReal:=Device.AO[4];
Device.TX.CH4[0]:=Data.tWord[0];
Device.TX.CH4[1]:=Data.tWord[1];


//Device.DSO.StrNamur:=Burkert_OSCAT_BASIC.REPLACE_ALL(str:=TO_STRING(Device.DSO.NamurNe107.eNamur) , src:='_' , rep:=' ' );

END_FUNCTION

// 20 Program Organization Units/Level_0_Remote_IO/eDip/eDip_ME44_DI
FUNCTION eDip_ME44_DI :BOOL;
VAR_INPUT
		device :REFERENCE TO ceDip_ME44_DI;
		Node:BYTE;
END_VAR
VAR
	//Data:Bytes_Dword;
END_VAR

Device.DSO.Node:=Node;
Device.Namur.iNamur:=Device.RX.Namur.tByte[1];

Device.Ch[1].Hz_Count:=Device.RX.DI1_Float.tReal;
Device.Ch[2].Hz_Count:=Device.RX.DI2_Float.tReal;
Device.Ch[3].Hz_Count:=Device.RX.DI3_Float.tReal;
Device.Ch[4].Hz_Count:=Device.RX.DI4_Float.tReal;
Device.Ch[5].Hz_Count:=Device.RX.DI5_Float.tReal;
Device.Ch[6].Hz_Count:=Device.RX.DI6_Float.tReal;
Device.Ch[7].Hz_Count:=Device.RX.DI7_Float.tReal;
Device.Ch[8].Hz_Count:=Device.RX.DI8_Float.tReal;

Device.Ch[1].Totaliser:=Device.RX.DI1_Total.tReal;
Device.Ch[2].Totaliser:=Device.RX.DI2_Total.tReal;
Device.Ch[3].Totaliser:=Device.RX.DI3_Total.tReal;
Device.Ch[4].Totaliser:=Device.RX.DI4_Total.tReal;
Device.Ch[5].Totaliser:=Device.RX.DI5_Total.tReal;
Device.Ch[6].Totaliser:=Device.RX.DI6_Total.tReal;
Device.Ch[7].Totaliser:=Device.RX.DI7_Total.tReal;
Device.Ch[8].Totaliser:=Device.RX.DI8_Total.tReal;

Device.Ch[1].Raw:=Device.RX.DI1_DI_8.tByte[1].0;
Device.Ch[2].Raw:=Device.RX.DI1_DI_8.tByte[1].1;
Device.Ch[3].Raw:=Device.RX.DI1_DI_8.tByte[1].2;
Device.Ch[4].Raw:=Device.RX.DI1_DI_8.tByte[1].3;
Device.Ch[5].Raw:=Device.RX.DI1_DI_8.tByte[1].4;
Device.Ch[6].Raw:=Device.RX.DI1_DI_8.tByte[1].5;
Device.Ch[7].Raw:=Device.RX.DI1_DI_8.tByte[1].6;
Device.Ch[8].Raw:=Device.RX.DI1_DI_8.tByte[1].7;





Device.TX.Counter_Reset.8:=Device.Ch[1].Reset_Count;
Device.TX.Totaliser_Reset.8:=Device.Ch[1].Reset_Totaliser;

Device.TX.Counter_Reset.9:=Device.Ch[2].Reset_Count;
Device.TX.Totaliser_Reset.9:=Device.Ch[2].Reset_Totaliser;

Device.TX.Counter_Reset.10:=Device.Ch[3].Reset_Count;
Device.TX.Totaliser_Reset.10:=Device.Ch[3].Reset_Totaliser;

Device.TX.Counter_Reset.11:=Device.Ch[4].Reset_Count;
Device.TX.Totaliser_Reset.11:=Device.Ch[4].Reset_Totaliser;

Device.TX.Counter_Reset.12:=Device.Ch[5].Reset_Count;
Device.TX.Totaliser_Reset.12:=Device.Ch[5].Reset_Totaliser;

Device.TX.Counter_Reset.13:=Device.Ch[6].Reset_Count;
Device.TX.Totaliser_Reset.13:=Device.Ch[6].Reset_Totaliser;

Device.TX.Counter_Reset.14:=Device.Ch[7].Reset_Count;
Device.TX.Totaliser_Reset.14:=Device.Ch[7].Reset_Totaliser;

Device.TX.Counter_Reset.15:=Device.Ch[8].Reset_Count;
Device.TX.Totaliser_Reset.15:=Device.Ch[8].Reset_Totaliser;

Device.DSO.StrNamur:=Burkert_OSCAT_BASIC.REPLACE_ALL(str:=TO_STRING(Device.DSO.NamurNe107.eNamur) , src:='_' , rep:=' ' );



device.Ready:=NOT((Device.Namur.eNamur=eNamur107.Error) OR (Device.Namur.eNamur=eNamur107.Offline));

END_FUNCTION

// 20 Program Organization Units/Level_0_Remote_IO/eDip/eDip_ME44_DO_Analog
FUNCTION eDip_ME44_DO_Analog : bool
VAR_INPUT
	Device: REFERENCE TO cME44_DO;
	DO_1:BOOL;
	DO_2:BOOL;
	DO_3:BOOL;
	DO_4:BOOL;
	DO_5:BOOL;
	DO_6:BOOL;
	DO_7:BOOL;
	DO_8:BOOL;
	
	PWM_1:REAL;
	PWM_2:REAL;
	PWM_3:REAL;
	PWM_4:REAL;
	PWM_5:REAL;
	PWM_6:REAL;
	PWM_7:REAL;
	PWM_8:REAL;
	
	
	
END_VAR
VAR
	Data:Bytes_Dword;
END_VAR

Data.tWord[0]:=Device.RX_Namur;
Device.Namur.iNamur:=Data.tByte[1];

Device.TX.CH1Ch8.8:=DO_1;
Device.TX.CH1Ch8.9:=DO_2;
Device.TX.CH1Ch8.10:=DO_3;
Device.TX.CH1Ch8.11:=DO_4;
Device.TX.CH1Ch8.12:=DO_5;
Device.TX.CH1Ch8.13:=DO_6;
Device.TX.CH1Ch8.14:=DO_7;
Device.TX.CH1Ch8.15:=DO_8;


Device.TX.CH1Bin.8:=DO_1;
Device.TX.CH2Bin.8:=DO_2;
Device.TX.CH3Bin.8:=DO_3;
Device.TX.CH4Bin.8:=DO_4;
Device.TX.CH5Bin.8:=DO_5;
Device.TX.CH6Bin.8:=DO_6;
Device.TX.CH7Bin.8:=DO_7;
Device.TX.CH8Bin.8:=DO_8;


Data.tReal:=PWM_1;
Device.TX.CH1Float[0]:=Data.tWord[0];
Device.TX.CH1Float[1]:=Data.tWord[1];

Data.tReal:=PWM_2;
Device.TX.CH2Float[0]:=Data.tWord[0];
Device.TX.CH2Float[1]:=Data.tWord[1];

Data.tReal:=PWM_3;
Device.TX.CH3Float[0]:=Data.tWord[0];
Device.TX.CH3Float[1]:=Data.tWord[1];

Data.tReal:=PWM_4;
Device.TX.CH4Float[0]:=Data.tWord[0];
Device.TX.CH4Float[1]:=Data.tWord[1];

Data.tReal:=PWM_5;
Device.TX.CH5Float[0]:=Data.tWord[0];
Device.TX.CH5Float[1]:=Data.tWord[1];

Data.tReal:=PWM_6;
Device.TX.CH6Float[0]:=Data.tWord[0];
Device.TX.CH6Float[1]:=Data.tWord[1];

Data.tReal:=PWM_7;
Device.TX.CH7Float[0]:=Data.tWord[0];
Device.TX.CH7Float[1]:=Data.tWord[1];

Data.tReal:=PWM_8;
Device.TX.CH8Float[0]:=Data.tWord[0];
Device.TX.CH8Float[1]:=Data.tWord[1];

//Device.DSO.StrNamur:=Burkert_OSCAT_BASIC.REPLACE_ALL(str:=TO_STRING(Device.DSO.NamurNe107.eNamur) , src:='_' , rep:=' ' );

END_FUNCTION

// 20 Program Organization Units/Level_0_Remote_IO/eDip/eDip_ME44_DO
FUNCTION eDip_ME44_DO : bool
VAR_INPUT
	Device: REFERENCE TO cME44_DO;
	DO_1:BOOL;
	DO_2:BOOL;
	DO_3:BOOL;
	DO_4:BOOL;
	DO_5:BOOL;
	DO_6:BOOL;
	DO_7:BOOL;
	DO_8:BOOL;
	
	
END_VAR
VAR
	Data:Bytes_Dword;
END_VAR

Data.tWord[0]:=Device.RX_Namur;
Device.Namur.iNamur:=Data.tByte[1];

Device.TX.CH1Ch8.8:=DO_1;
Device.TX.CH1Ch8.9:=DO_2;
Device.TX.CH1Ch8.10:=DO_3;
Device.TX.CH1Ch8.11:=DO_4;
Device.TX.CH1Ch8.12:=DO_5;
Device.TX.CH1Ch8.13:=DO_6;
Device.TX.CH1Ch8.14:=DO_7;
Device.TX.CH1Ch8.15:=DO_8;


Device.TX.CH1Bin.8:=DO_1;
Device.TX.CH2Bin.8:=DO_2;
Device.TX.CH3Bin.8:=DO_3;
Device.TX.CH4Bin.8:=DO_4;
Device.TX.CH5Bin.8:=DO_5;
Device.TX.CH6Bin.8:=DO_6;
Device.TX.CH7Bin.8:=DO_7;
Device.TX.CH8Bin.8:=DO_8;


//Device.DSO.StrNamur:=Burkert_OSCAT_BASIC.REPLACE_ALL(str:=TO_STRING(Device.DSO.NamurNe107.eNamur) , src:='_' , rep:=' ' );

END_FUNCTION

// 20 Program Organization Units/Level_0_Remote_IO/eDip/Parse_DDO
FUNCTION_BLOCK Parse_DDO
VAR_INPUT
	ORF_data:POINTER TO BYTE;
	Node:BYTE;
	Request_Size:INT:=10;
	
END_VAR
VAR_OUTPUT
	DDO:eDip_DDO;
END_VAR
VAR
	Block_Size:UINT;
	lcl_pointer:POINTER TO BYTE;
	DDO_Index:INT;
	ORF_Node:BYTE;
	ORF_Index_HB:BYTE;
	ORF_Index_LB:BYTE;
	ORF_SubIndex:BYTE;
	
	
END_VAR

Block_Size:=SIZEOF(ORF_Request);
lcl_pointer:=ORF_Data;

FOR DDO_Index := 0 TO Request_Size BY 1 DO
	
	ORF_Index_LB:=lcl_pointer[0];
	ORF_Index_HB:=LCL_Pointer[1];
	ORF_SubIndex:=lcl_pointer[2];
	ORF_Node:=lcl_pointer[3];
	
	
	IF (lcl_pointer[10]=1) AND (ORF_Node= Node) AND (ORF_Index_HB=16#20) AND (ORF_Index_LB=16#00) THEN
		MEMUtils.MemSet(pbyBuffer:=lcl_pointer+10 , byValue:=0 , dwSize:= 1); // Clear Complete
		CASE ORF_SubIndex OF
			16#02: //16#2000-2
				MEMUtils.MemCpy(pbyDest:=ADR(DDO.Ident)+2 , pbySrc:=lcl_pointer+4 , dwSize:=2 );
				MEMUtils.MemCpy(pbyDest:=ADR(DDO.Ident) , pbySrc:=lcl_pointer+6 , dwSize:=2 );
				lcl_pointer[9]:=BOOL_TO_BYTE(DDO.Ident=0);
				//MEMUtils.MemSet(pbyBuffer:=lcl_pointer+9 , byValue:=1 , dwSize:= 1);// Set Enable				
			16#07: //16#2000-7
				MEMUtils.MemCpy(pbyDest:=ADR(DDO.Serial)+2 , pbySrc:=lcl_pointer+4 , dwSize:=2 );
				MEMUtils.MemCpy(pbyDest:=ADR(DDO.Serial) , pbySrc:=lcl_pointer+6 , dwSize:=2 );
				lcl_pointer[9]:=BOOL_TO_BYTE(DDO.Serial=0);
			16#008: //16#2000-8
				MEMUtils.MemCpy(pbyDest:=ADR(DDO.Product_Code)+2 , pbySrc:=lcl_pointer+4 , dwSize:=2 );
				MEMUtils.MemCpy(pbyDest:=ADR(DDO.Product_Code) , pbySrc:=lcl_pointer+6 , dwSize:=2 );
				lcl_pointer[9]:=BOOL_TO_BYTE(DDO.Product_Code =0);
		END_CASE;	
	END_IF;
	lcl_pointer:=lcl_pointer+Block_Size;
END_FOR;

END_FUNCTION_BLOCK

// 20 Program Organization Units/Level_0_Remote_IO/eDip/Parse_DSO
FUNCTION_BLOCK Parse_DSO
VAR_INPUT
	ORF_data:POINTER TO BYTE;
	Node:BYTE;
	Request_Size:INT:=10;
	
END_VAR
VAR_OUTPUT
	DSO:eDip_DSO;
END_VAR
VAR
	Block_Size:UINT;
	lcl_pointer:POINTER TO BYTE;
	DSO_Index:INT;
	ORF_Node:BYTE;
	ORF_Index_HB:BYTE;
	ORF_Index_LB:BYTE;
	ORF_SubIndex:BYTE;
	
END_VAR

Block_Size:=SIZEOF(ORF_Request);
lcl_pointer:=ORF_Data;

FOR DSO_Index := 0 TO Request_Size BY 1 DO
	ORF_Index_LB:=lcl_pointer[0];
	ORF_Index_HB:=LCL_Pointer[1];
	ORF_SubIndex:=lcl_pointer[2];
	ORF_Node:=lcl_pointer[3];
	
	IF (lcl_pointer[10]=1) AND (ORF_Node= Node) AND (ORF_Index_HB=16#20) AND (ORF_Index_LB=16#04) THEN
		//MEMUtils.MemSet(pbyBuffer:=lcl_pointer+10 , byValue:=0 , dwSize:= 1); // Clear Complete
		lcl_pointer[10]:=0;
		CASE ORF_SubIndex OF
			
